LIN {X 0,Y 448.603,Z 481.559,A -85,B 0,C 180,E1 -8747.553,E2 -8747.553} C_VEL
LIN {X 0,Y 449.563,Z 469.193,A -85,B 0,C 180,E1 -8748.693,E2 -8748.693} C_VEL
LIN {X 0,Y 450.592,Z 455.729,A -85,B 0,C 180,E1 -8749.713,E2 -8749.713} C_VEL
LIN {X 0,Y 451.602,Z 440.797,A -85,B 0,C 180,E1 -8750.617,E2 -8750.617} C_VEL
LIN {X 0,Y 452.485,Z 425.824,A -85,B 0,C 180,E1 -8751.309,E2 -8751.309} C_VEL
LIN {X 0,Y 453.202,Z 410.38,A -85,B 0,C 180,E1 -8751.823,E2 -8751.823} C_VEL
LIN {X 0,Y 453.655,Z 394.686,A -85,B 0,C 180,E1 -8752.157,E2 -8752.157} C_VEL
LIN {X 0,Y 455.333,Z 264.862,A -85,B 0,C 180,E1 -8754.24,E2 -8754.24} C_VEL
LIN {X 0,Y 453.979,Z 251.014,A -85,B 0,C 180,E1 -8754.549,E2 -8754.549} C_VEL
LIN {X 0,Y 452.072,Z 236.66,A -85,B 0,C 180,E1 -8754.969,E2 -8754.969} C_VEL
LIN {X 0,Y 454.282,Z 211.093,A -85,B 0,C 180,E1 -8757.828,E2 -8757.828} C_VEL
LIN {X 0,Y 457.111,Z 186.417,A -85,B 0,C 180,E1 -8760.745,E2 -8760.745} C_VEL
LIN {X 0,Y 457.91,Z 180.659,A -85,B 0,C 180,E1 -8761.456,E2 -8761.456} C_VEL
LIN {X 0,Y 455.867,Z 172.549,A -85,B 0,C 180,E1 -8762.832,E2 -8762.832} C_VEL
LIN {X 0,Y 452.903,Z 163.172,A -85,B 0,C 180,E1 -8764.671,E2 -8764.671} C_VEL
LIN {X 0,Y 449.695,Z 154.889,A -85,B 0,C 180,E1 -8766.634,E2 -8766.634} C_VEL
LIN {X 0,Y 447.386,Z 149.256,A -85,B 0,C 180,E1 -8768.238,E2 -8768.238} C_VEL
LIN {X 0,Y 446.421,Z 146.504,A -85,B 0,C 180,E1 -8769.151,E2 -8769.151} C_VEL
LIN {X 0,Y 446.382,Z 146.509,A -85,B 0,C 180,E1 -8772.27,E2 -8772.27} C_VEL
LIN {X 0,Y 446.423,Z 146.505,A -85,B 0,C 180,E1 -8775.108,E2 -8775.108} C_VEL
LIN {X 0,Y 446.397,Z 146.505,A -85,B 0,C 180,E1 -8778.606,E2 -8778.606} C_VEL
LIN {X 0,Y 446.39,Z 146.508,A -85,B 0,C 180,E1 -8782.119,E2 -8782.119} C_VEL
LIN {X 0,Y 446.423,Z 146.505,A -85,B 0,C 180,E1 -8785.477,E2 -8785.477} C_VEL
LIN {X 0,Y 446.442,Z 146.59,A -85,B 0,C 180,E1 -8786.407,E2 -8786.407} C_VEL
LIN {X 0,Y 448.873,Z 153.492,A -85,B 0,C 180,E1 -8788.89,E2 -8788.89} C_VEL
LIN {X 0,Y 451.118,Z 160.8,A -85,B 0,C 180,E1 -8791.122,E2 -8791.122} C_VEL
LIN {X 0,Y 453.267,Z 168.747,A -85,B 0,C 180,E1 -8793.279,E2 -8793.279} C_VEL
LIN {X 0,Y 454.691,Z 176.225,A -85,B 0,C 180,E1 -8795.09,E2 -8795.09} C_VEL
LIN {X 0,Y 453.323,Z 189.363,A -85,B 0,C 180,E1 -8797.677,E2 -8797.677} C_VEL
LIN {X 0,Y 451.857,Z 205.223,A -85,B 0,C 180,E1 -8800.671,E2 -8800.671} C_VEL
LIN {X 0,Y 455.219,Z 218.827,A -85,B 0,C 180,E1 -8801.302,E2 -8801.302} C_VEL
LIN {X 0,Y 451.899,Z 307.293,A -85,B 0,C 180,E1 -8803.453,E2 -8803.453} C_VEL
LIN {X 0,Y 451.558,Z 325.184,A -85,B 0,C 180,E1 -8803.934,E2 -8803.934} C_VEL
LIN {X 0,Y 451.243,Z 338.258,A -85,B 0,C 180,E1 -8804.473,E2 -8804.473} C_VEL
LIN {X 0,Y 450.777,Z 351.293,A -85,B 0,C 180,E1 -8805.198,E2 -8805.198} C_VEL
LIN {X 0,Y 450.232,Z 362.94,A -85,B 0,C 180,E1 -8806.028,E2 -8806.028} C_VEL
LIN {X 0,Y 449.679,Z 373.95,A -85,B 0,C 180,E1 -8807.017,E2 -8807.017} C_VEL
LIN {X 0,Y 449.213,Z 383.222,A -85,B 0,C 180,E1 -8808.036,E2 -8808.036} C_VEL
LIN {X 0,Y 448.662,Z 391.778,A -85,B 0,C 180,E1 -8809.166,E2 -8809.166} C_VEL
LIN {X 0,Y 448.106,Z 400.134,A -85,B 0,C 180,E1 -8810.521,E2 -8810.521} C_VEL
LIN {X 0,Y 447.566,Z 406.817,A -85,B 0,C 180,E1 -8811.876,E2 -8811.876} C_VEL
LIN {X 0,Y 447.282,Z 412.123,A -85,B 0,C 180,E1 -8813.232,E2 -8813.232} C_VEL
LIN {X 0,Y 446.899,Z 416.261,A -85,B 0,C 180,E1 -8814.586,E2 -8814.586} C_VEL
LIN {X 0,Y 446.735,Z 418.408,A -85,B 0,C 180,E1 -8815.489,E2 -8815.489} C_VEL
LIN {X 0,Y 446.7,Z 420.094,A -85,B 0,C 180,E1 -8816.392,E2 -8816.392} C_VEL
LIN {X 0,Y 446.587,Z 421.324,A -85,B 0,C 180,E1 -8817.294,E2 -8817.294} C_VEL
LIN {X 0,Y 446.509,Z 422.142,A -85,B 0,C 180,E1 -8818.196,E2 -8818.196} C_VEL
LIN {X 0,Y 446.414,Z 422.565,A -85,B 0,C 180,E1 -8819.098,E2 -8819.098} C_VEL
LIN {X 0,Y 446.372,Z 422.567,A -85,B 0,C 180,E1 -8820,E2 -8820} C_VEL
LIN {X 0,Y 446.387,Z 422.116,A -85,B 0,C 180,E1 -8820.902,E2 -8820.902} C_VEL
LIN {X 0,Y 446.305,Z 421.284,A -85,B 0,C 180,E1 -8821.805,E2 -8821.805} C_VEL
LIN {X 0,Y 446.422,Z 420.025,A -85,B 0,C 180,E1 -8822.707,E2 -8822.707} C_VEL
LIN {X 0,Y 446.362,Z 417.34,A -85,B 0,C 180,E1 -8824.063,E2 -8824.063} C_VEL
LIN {X 0,Y 446.544,Z 413.61,A -85,B 0,C 180,E1 -8825.419,E2 -8825.419} C_VEL
LIN {X 0,Y 446.83,Z 408.619,A -85,B 0,C 180,E1 -8826.811,E2 -8826.811} C_VEL
LIN {X 0,Y 447.019,Z 402.697,A -85,B 0,C 180,E1 -8828.135,E2 -8828.135} C_VEL
LIN {X 0,Y 447.423,Z 395.107,A -85,B 0,C 180,E1 -8829.493,E2 -8829.493} C_VEL
LIN {X 0,Y 447.76,Z 385.722,A -85,B 0,C 180,E1 -8830.857,E2 -8830.857} C_VEL
LIN {X 0,Y 448.163,Z 376.127,A -85,B 0,C 180,E1 -8831.993,E2 -8831.993} C_VEL
LIN {X 0,Y 448.646,Z 365.513,A -85,B 0,C 180,E1 -8833.014,E2 -8833.014} C_VEL
LIN {X 0,Y 449.076,Z 352.8,A -85,B 0,C 180,E1 -8833.998,E2 -8833.998} C_VEL
LIN {X 0,Y 449.421,Z 340.82,A -85,B 0,C 180,E1 -8834.721,E2 -8834.721} C_VEL
LIN {X 0,Y 449.721,Z 326.89,A -85,B 0,C 180,E1 -8835.349,E2 -8835.349} C_VEL
LIN {X 0,Y 449.994,Z 313.038,A -85,B 0,C 180,E1 -8835.775,E2 -8835.775} C_VEL
LIN {X 0,Y 451.496,Z 214.96,A -85,B 0,C 180,E1 -8837.673,E2 -8837.673} C_VEL
LIN {X 0,Y 448.658,Z 199.549,A -85,B 0,C 180,E1 -8838.105,E2 -8838.105} C_VEL
LIN {X 0,Y 449.604,Z 180.934,A -85,B 0,C 180,E1 -8841.311,E2 -8841.311} C_VEL
LIN {X 0,Y 450.318,Z 165.889,A -85,B 0,C 180,E1 -8843.94,E2 -8843.94} C_VEL
LIN {X 0,Y 449.539,Z 160.406,A -85,B 0,C 180,E1 -8844.968,E2 -8844.968} C_VEL
LIN {X 0,Y 446.472,Z 146.498,A -85,B 0,C 180,E1 -8847.7,E2 -8847.7} C_VEL
LIN {X 0,Y 446.431,Z 146.5,A -85,B 0,C 180,E1 -8850.25,E2 -8850.25} C_VEL
LIN {X 0,Y 446.451,Z 146.501,A -85,B 0,C 180,E1 -8853.453,E2 -8853.453} C_VEL
LIN {X 0,Y 446.405,Z 146.503,A -85,B 0,C 180,E1 -8856.745,E2 -8856.745} C_VEL
LIN {X 0,Y 446.44,Z 146.491,A -85,B 0,C 180,E1 -8860.198,E2 -8860.198} C_VEL
LIN {X 0,Y 446.402,Z 146.498,A -85,B 0,C 180,E1 -8863.596,E2 -8863.596} C_VEL
LIN {X 0,Y 446.403,Z 146.503,A -85,B 0,C 180,E1 -8866.403,E2 -8866.403} C_VEL
LIN {X 0,Y 446.432,Z 146.501,A -85,B 0,C 180,E1 -8869.082,E2 -8869.082} C_VEL
LIN {X 0,Y 446.413,Z 146.503,A -85,B 0,C 180,E1 -8872.121,E2 -8872.121} C_VEL
LIN {X 0,Y 446.427,Z 146.503,A -85,B 0,C 180,E1 -8875.476,E2 -8875.476} C_VEL
LIN {X 0,Y 446.42,Z 146.503,A -85,B 0,C 180,E1 -8878.699,E2 -8878.699} C_VEL
LIN {X 0,Y 446.494,Z 146.615,A -85,B 0,C 180,E1 -8881.866,E2 -8881.866} C_VEL
LIN {X 0,Y 449.989,Z 159.891,A -85,B 0,C 180,E1 -8884.067,E2 -8884.067} C_VEL
LIN {X 0,Y 451.233,Z 164.799,A -85,B 0,C 180,E1 -8884.784,E2 -8884.784} C_VEL
LIN {X 0,Y 454.277,Z 173.036,A -85,B 0,C 180,E1 -8885.111,E2 -8885.111} C_VEL
LIN {X 0,Y 456.804,Z 184.373,A -85,B 0,C 180,E1 -8885.455,E2 -8885.455} C_VEL
LIN {X 0,Y 456.787,Z 190.412,A -85,B 0,C 180,E1 -8885.557,E2 -8885.557} C_VEL
LIN {X 0,Y 456.125,Z 196.262,A -85,B 0,C 180,E1 -8885.618,E2 -8885.618} C_VEL
LIN {X 0,Y 450.604,Z 215.327,A -85,B 0,C 180,E1 -8885.621,E2 -8885.621} C_VEL
LIN {X 0,Y 449.88,Z 221.18,A -85,B 0,C 180,E1 -8885.68,E2 -8885.68} C_VEL
LIN {X 0,Y 448.241,Z 331.634,A -85,B 0,C 180,E1 -8887.512,E2 -8887.512} C_VEL
LIN {X 0,Y 447.916,Z 346.746,A -85,B 0,C 180,E1 -8887.937,E2 -8887.937} C_VEL
LIN {X 0,Y 447.417,Z 359.567,A -85,B 0,C 180,E1 -8888.442,E2 -8888.442} C_VEL
LIN {X 0,Y 446.764,Z 373.298,A -85,B 0,C 180,E1 -8889.15,E2 -8889.15} C_VEL
LIN {X 0,Y 445.828,Z 387.352,A -85,B 0,C 180,E1 -8890.068,E2 -8890.068} C_VEL
LIN {X 0,Y 444.831,Z 400.144,A -85,B 0,C 180,E1 -8891.101,E2 -8891.101} C_VEL
LIN {X 0,Y 443.852,Z 412.557,A -85,B 0,C 180,E1 -8892.325,E2 -8892.325} C_VEL
LIN {X 0,Y 442.838,Z 423.693,A -85,B 0,C 180,E1 -8893.637,E2 -8893.637} C_VEL
LIN {X 0,Y 441.963,Z 433.554,A -85,B 0,C 180,E1 -8895.024,E2 -8895.024} C_VEL
LIN {X 0,Y 441.073,Z 442.905,A -85,B 0,C 180,E1 -8896.59,E2 -8896.59} C_VEL
LIN {X 0,Y 440.345,Z 451.156,A -85,B 0,C 180,E1 -8898.258,E2 -8898.258} C_VEL
LIN {X 0,Y 439.756,Z 457.752,A -85,B 0,C 180,E1 -8899.874,E2 -8899.874} C_VEL
LIN {X 0,Y 439.297,Z 463.848,A -85,B 0,C 180,E1 -8901.72,E2 -8901.72} C_VEL
LIN {X 0,Y 438.938,Z 468.563,A -85,B 0,C 180,E1 -8903.564,E2 -8903.564} C_VEL
LIN {X 0,Y 438.817,Z 472.01,A -85,B 0,C 180,E1 -8905.406,E2 -8905.406} C_VEL
LIN {X 0,Y 438.65,Z 474.293,A -85,B 0,C 180,E1 -8907.244,E2 -8907.244} C_VEL
LIN {X 0,Y 438.422,Z 475.467,A -85,B 0,C 180,E1 -8909.08,E2 -8909.08} C_VEL
LIN {X 0,Y 438.422,Z 475.482,A -85,B 0,C 180,E1 -8910.917,E2 -8910.917} C_VEL
LIN {X 0,Y 438.649,Z 474.369,A -85,B 0,C 180,E1 -8912.754,E2 -8912.754} C_VEL
LIN {X 0,Y 438.808,Z 472.151,A -85,B 0,C 180,E1 -8914.592,E2 -8914.592} C_VEL
LIN {X 0,Y 438.92,Z 468.778,A -85,B 0,C 180,E1 -8916.434,E2 -8916.434} C_VEL
LIN {X 0,Y 439.284,Z 464.136,A -85,B 0,C 180,E1 -8918.277,E2 -8918.277} C_VEL
LIN {X 0,Y 439.743,Z 458.109,A -85,B 0,C 180,E1 -8920.124,E2 -8920.124} C_VEL
LIN {X 0,Y 440.383,Z 450.519,A -85,B 0,C 180,E1 -8921.973,E2 -8921.973} C_VEL
LIN {X 0,Y 441.164,Z 442.089,A -85,B 0,C 180,E1 -8923.647,E2 -8923.647} C_VEL
LIN {X 0,Y 442.056,Z 432.628,A -85,B 0,C 180,E1 -8925.207,E2 -8925.207} C_VEL
LIN {X 0,Y 442.961,Z 422.624,A -85,B 0,C 180,E1 -8926.593,E2 -8926.593} C_VEL
LIN {X 0,Y 443.984,Z 410.668,A -85,B 0,C 180,E1 -8927.973,E2 -8927.973} C_VEL
LIN {X 0,Y 444.997,Z 398.609,A -85,B 0,C 180,E1 -8929.129,E2 -8929.129} C_VEL
LIN {X 0,Y 446.011,Z 385.476,A -85,B 0,C 180,E1 -8930.162,E2 -8930.162} C_VEL
LIN {X 0,Y 446.863,Z 370.893,A -85,B 0,C 180,E1 -8931.084,E2 -8931.084} C_VEL
LIN {X 0,Y 447.531,Z 356.049,A -85,B 0,C 180,E1 -8931.81,E2 -8931.81} C_VEL
LIN {X 0,Y 448.081,Z 341.166,A -85,B 0,C 180,E1 -8932.338,E2 -8932.338} C_VEL
LIN {X 0,Y 448.349,Z 327.58,A -85,B 0,C 180,E1 -8932.668,E2 -8932.668} C_VEL
LIN {X 0,Y 450.438,Z 185.764,A -85,B 0,C 180,E1 -8934.996,E2 -8934.996} C_VEL
LIN {X 0,Y 447.373,Z 172.856,A -85,B 0,C 180,E1 -8935.409,E2 -8935.409} C_VEL
LIN {X 0,Y 444.02,Z 164.852,A -85,B 0,C 180,E1 -8935.791,E2 -8935.791} C_VEL
LIN {X 0,Y 440.796,Z 152.391,A -85,B 0,C 180,E1 -8937.774,E2 -8937.774} C_VEL
LIN {X 0,Y 439.435,Z 147.373,A -85,B 0,C 180,E1 -8938.671,E2 -8938.671} C_VEL
LIN {X 0,Y 439.366,Z 147.373,A -85,B 0,C 180,E1 -8942.029,E2 -8942.029} C_VEL
LIN {X 0,Y 439.391,Z 147.38,A -85,B 0,C 180,E1 -8945.339,E2 -8945.339} C_VEL
LIN {X 0,Y 439.377,Z 147.377,A -85,B 0,C 180,E1 -8948.594,E2 -8948.594} C_VEL
LIN {X 0,Y 439.383,Z 147.367,A -85,B 0,C 180,E1 -8951.256,E2 -8951.256} C_VEL
LIN {X 0,Y 439.398,Z 147.37,A -85,B 0,C 180,E1 -8954.727,E2 -8954.727} C_VEL
LIN {X 0,Y 439.39,Z 147.374,A -85,B 0,C 180,E1 -8957.795,E2 -8957.795} C_VEL
LIN {X 0,Y 439.444,Z 147.367,A -85,B 0,C 180,E1 -8960.229,E2 -8960.229} C_VEL
LIN {X 0,Y 439.369,Z 147.378,A -85,B 0,C 180,E1 -8963.712,E2 -8963.712} C_VEL
LIN {X 0,Y 439.367,Z 147.38,A -85,B 0,C 180,E1 -8967.053,E2 -8967.053} C_VEL
LIN {X 0,Y 439.388,Z 147.365,A -85,B 0,C 180,E1 -8970.274,E2 -8970.274} C_VEL
LIN {X 0,Y 439.423,Z 147.369,A -85,B 0,C 180,E1 -8973.588,E2 -8973.588} C_VEL
LIN {X 0,Y 439.376,Z 147.372,A -85,B 0,C 180,E1 -8976.429,E2 -8976.429} C_VEL
LIN {X 0,Y 439.378,Z 147.373,A -85,B 0,C 180,E1 -8979.396,E2 -8979.396} C_VEL
LIN {X 0,Y 439.421,Z 147.366,A -85,B 0,C 180,E1 -8982.309,E2 -8982.309} C_VEL
LIN {X 0,Y 439.438,Z 147.367,A -85,B 0,C 180,E1 -8985.174,E2 -8985.174} C_VEL
LIN {X 0,Y 439.474,Z 147.356,A -85,B 0,C 180,E1 -8988.001,E2 -8988.001} C_VEL
LIN {X 0,Y 439.537,Z 147.353,A -85,B 0,C 180,E1 -8991.726,E2 -8991.726} C_VEL
LIN {X 0,Y 439.61,Z 147.338,A -85,B 0,C 180,E1 -8994.496,E2 -8994.496} C_VEL
LIN {X 0,Y 439.625,Z 147.346,A -85,B 0,C 180,E1 -8998.168,E2 -8998.168} C_VEL
LIN {X 0,Y 439.753,Z 147.319,A -85,B 0,C 180,E1 -9000,E2 -9000} C_VEL
LIN {X 0,Y 439.646,Z 147.347,A -85,B 0,C 180,E1 -9002.749,E2 -9002.749} C_VEL
LIN {X 0,Y 439.607,Z 147.338,A -85,B 0,C 180,E1 -9006.425,E2 -9006.425} C_VEL
LIN {X 0,Y 439.49,Z 147.36,A -85,B 0,C 180,E1 -9009.202,E2 -9009.202} C_VEL
LIN {X 0,Y 439.455,Z 147.355,A -85,B 0,C 180,E1 -9012.938,E2 -9012.938} C_VEL
LIN {X 0,Y 439.449,Z 147.37,A -85,B 0,C 180,E1 -9016.355,E2 -9016.355} C_VEL
LIN {X 0,Y 439.393,Z 147.364,A -85,B 0,C 180,E1 -9019.627,E2 -9019.627} C_VEL
LIN {X 0,Y 439.357,Z 147.379,A -85,B 0,C 180,E1 -9022.576,E2 -9022.576} C_VEL
LIN {X 0,Y 439.395,Z 147.369,A -85,B 0,C 180,E1 -9025.585,E2 -9025.585} C_VEL
LIN {X 0,Y 439.407,Z 147.368,A -85,B 0,C 180,E1 -9028.674,E2 -9028.674} C_VEL
LIN {X 0,Y 439.361,Z 147.382,A -85,B 0,C 180,E1 -9032.031,E2 -9032.031} C_VEL
LIN {X 0,Y 439.387,Z 147.373,A -85,B 0,C 180,E1 -9035.342,E2 -9035.342} C_VEL
LIN {X 0,Y 439.379,Z 147.364,A -85,B 0,C 180,E1 -9038.595,E2 -9038.595} C_VEL
LIN {X 0,Y 439.379,Z 147.359,A -85,B 0,C 180,E1 -9041.258,E2 -9041.258} C_VEL
LIN {X 0,Y 439.394,Z 147.376,A -85,B 0,C 180,E1 -9044.73,E2 -9044.73} C_VEL
LIN {X 0,Y 439.405,Z 147.377,A -85,B 0,C 180,E1 -9047.799,E2 -9047.799} C_VEL
LIN {X 0,Y 439.442,Z 147.372,A -85,B 0,C 180,E1 -9050.231,E2 -9050.231} C_VEL
LIN {X 0,Y 439.37,Z 147.376,A -85,B 0,C 180,E1 -9053.714,E2 -9053.714} C_VEL
LIN {X 0,Y 439.393,Z 147.429,A -85,B 0,C 180,E1 -9054.55,E2 -9054.55} C_VEL
LIN {X 0,Y 445.757,Z 168.464,A -85,B 0,C 180,E1 -9057.489,E2 -9057.489} C_VEL
LIN {X 0,Y 448.797,Z 178.964,A -85,B 0,C 180,E1 -9058.886,E2 -9058.886} C_VEL
LIN {X 0,Y 446.1,Z 212.955,A -85,B 0,C 180,E1 -9062.562,E2 -9062.562} C_VEL
LIN {X 0,Y 444.881,Z 231.94,A -85,B 0,C 180,E1 -9064.588,E2 -9064.588} C_VEL
LIN {X 0,Y 448.797,Z 263.831,A -85,B 0,C 180,E1 -9065.369,E2 -9065.369} C_VEL
LIN {X 0,Y 447.227,Z 382.055,A -85,B 0,C 180,E1 -9067.296,E2 -9067.296} C_VEL
LIN {X 0,Y 446.797,Z 404.556,A -85,B 0,C 180,E1 -9067.7,E2 -9067.7} C_VEL
LIN {X 0,Y 446.125,Z 419.902,A -85,B 0,C 180,E1 -9068.152,E2 -9068.152} C_VEL
LIN {X 0,Y 445.255,Z 434.727,A -85,B 0,C 180,E1 -9068.775,E2 -9068.775} C_VEL
LIN {X 0,Y 444.41,Z 448.229,A -85,B 0,C 180,E1 -9069.521,E2 -9069.521} C_VEL
LIN {X 0,Y 443.348,Z 461.563,A -85,B 0,C 180,E1 -9070.436,E2 -9070.436} C_VEL
LIN {X 0,Y 442.298,Z 475.142,A -85,B 0,C 180,E1 -9071.592,E2 -9071.592} C_VEL
LIN {X 0,Y 441.431,Z 486.843,A -85,B 0,C 180,E1 -9072.796,E2 -9072.796} C_VEL
LIN {X 0,Y 440.489,Z 498.759,A -85,B 0,C 180,E1 -9074.264,E2 -9074.264} C_VEL
LIN {X 0,Y 439.65,Z 509.698,A -85,B 0,C 180,E1 -9075.892,E2 -9075.892} C_VEL
LIN {X 0,Y 439.142,Z 518.621,A -85,B 0,C 180,E1 -9077.485,E2 -9077.485} C_VEL
LIN {X 0,Y 438.821,Z 527.349,A -85,B 0,C 180,E1 -9079.388,E2 -9079.388} C_VEL
LIN {X 0,Y 438.548,Z 534.198,A -85,B 0,C 180,E1 -9081.244,E2 -9081.244} C_VEL
LIN {X 0,Y 438.584,Z 539.573,A -85,B 0,C 180,E1 -9083.099,E2 -9083.099} C_VEL
LIN {X 0,Y 438.605,Z 542.66,A -85,B 0,C 180,E1 -9084.484,E2 -9084.484} C_VEL
LIN {X 0,Y 438.639,Z 545.687,A -85,B 0,C 180,E1 -9086.327,E2 -9086.327} C_VEL
LIN {X 0,Y 438.591,Z 547.489,A -85,B 0,C 180,E1 -9088.165,E2 -9088.165} C_VEL
LIN {X 0,Y 438.645,Z 548.109,A -85,B 0,C 180,E1 -9090.001,E2 -9090.001} C_VEL
LIN {X 0,Y 438.591,Z 547.489,A -85,B 0,C 180,E1 -9091.838,E2 -9091.838} C_VEL
LIN {X 0,Y 438.64,Z 545.687,A -85,B 0,C 180,E1 -9093.676,E2 -9093.676} C_VEL
LIN {X 0,Y 438.604,Z 542.653,A -85,B 0,C 180,E1 -9095.518,E2 -9095.518} C_VEL
LIN {X 0,Y 438.596,Z 538.327,A -85,B 0,C 180,E1 -9097.366,E2 -9097.366} C_VEL
LIN {X 0,Y 438.637,Z 532.608,A -85,B 0,C 180,E1 -9099.221,E2 -9099.221} C_VEL
LIN {X 0,Y 438.899,Z 525.353,A -85,B 0,C 180,E1 -9101.08,E2 -9101.08} C_VEL
LIN {X 0,Y 439.272,Z 517.378,A -85,B 0,C 180,E1 -9102.747,E2 -9102.747} C_VEL
LIN {X 0,Y 439.78,Z 508.222,A -85,B 0,C 180,E1 -9104.343,E2 -9104.343} C_VEL
LIN {X 0,Y 440.514,Z 498.723,A -85,B 0,C 180,E1 -9105.738,E2 -9105.738} C_VEL
LIN {X 0,Y 441.425,Z 486.832,A -85,B 0,C 180,E1 -9107.202,E2 -9107.202} C_VEL
LIN {X 0,Y 442.215,Z 476.257,A -85,B 0,C 180,E1 -9108.294,E2 -9108.294} C_VEL
LIN {X 0,Y 443.145,Z 464.364,A -85,B 0,C 180,E1 -9109.334,E2 -9109.334} C_VEL
LIN {X 0,Y 444.1,Z 451.678,A -85,B 0,C 180,E1 -9110.255,E2 -9110.255} C_VEL
LIN {X 0,Y 445.038,Z 437.98,A -85,B 0,C 180,E1 -9111.056,E2 -9111.056} C_VEL
LIN {X 0,Y 445.951,Z 423.205,A -85,B 0,C 180,E1 -9111.719,E2 -9111.719} C_VEL
LIN {X 0,Y 446.681,Z 408.798,A -85,B 0,C 180,E1 -9112.187,E2 -9112.187} C_VEL
LIN {X 0,Y 447.104,Z 392.425,A -85,B 0,C 180,E1 -9112.53,E2 -9112.53} C_VEL
LIN {X 0,Y 448.81,Z 263.796,A -85,B 0,C 180,E1 -9114.625,E2 -9114.625} C_VEL
LIN {X 0,Y 447.301,Z 249.61,A -85,B 0,C 180,E1 -9114.995,E2 -9114.995} C_VEL
LIN {X 0,Y 445.597,Z 236.028,A -85,B 0,C 180,E1 -9115.456,E2 -9115.456} C_VEL
LIN {X 0,Y 448.261,Z 208.763,A -85,B 0,C 180,E1 -9118.599,E2 -9118.599} C_VEL
LIN {X 0,Y 451.564,Z 183.576,A -85,B 0,C 180,E1 -9121.688,E2 -9121.688} C_VEL
LIN {X 0,Y 450.44,Z 178.248,A -85,B 0,C 180,E1 -9122.591,E2 -9122.591} C_VEL
LIN {X 0,Y 447.693,Z 168.89,A -85,B 0,C 180,E1 -9124.413,E2 -9124.413} C_VEL
LIN {X 0,Y 444.742,Z 160.784,A -85,B 0,C 180,E1 -9126.301,E2 -9126.301} C_VEL
LIN {X 0,Y 441.878,Z 153.645,A -85,B 0,C 180,E1 -9128.338,E2 -9128.338} C_VEL
LIN {X 0,Y 440.702,Z 150.674,A -85,B 0,C 180,E1 -9129.337,E2 -9129.337} C_VEL
LIN {X 0,Y 439.502,Z 148.11,A -85,B 0,C 180,E1 -9130.364,E2 -9130.364} C_VEL
LIN {X 0,Y 439.355,Z 147.384,A -85,B 0,C 180,E1 -9130.682,E2 -9130.682} C_VEL
LIN {X 0,Y 439.355,Z 147.385,A -85,B 0,C 180,E1 -9133.96,E2 -9133.96} C_VEL
LIN {X 0,Y 439.333,Z 147.385,A -85,B 0,C 180,E1 -9136.538,E2 -9136.538} C_VEL
LIN {X 0,Y 439.35,Z 147.385,A -85,B 0,C 180,E1 -9139.016,E2 -9139.016} C_VEL
LIN {X 0,Y 439.336,Z 147.386,A -85,B 0,C 180,E1 -9142.564,E2 -9142.564} C_VEL
LIN {X 0,Y 439.394,Z 147.383,A -85,B 0,C 180,E1 -9144.844,E2 -9144.844} C_VEL
LIN {X 0,Y 441.661,Z 153.659,A -85,B 0,C 180,E1 -9147.499,E2 -9147.499} C_VEL
LIN {X 0,Y 444.176,Z 161.248,A -85,B 0,C 180,E1 -9150.106,E2 -9150.106} C_VEL
LIN {X 0,Y 446.765,Z 170.807,A -85,B 0,C 180,E1 -9152.858,E2 -9152.858} C_VEL
LIN {X 0,Y 448.19,Z 178.084,A -85,B 0,C 180,E1 -9154.704,E2 -9154.704} C_VEL
LIN {X 0,Y 447.874,Z 182.864,A -85,B 0,C 180,E1 -9155.705,E2 -9155.705} C_VEL
LIN {X 0,Y 445.995,Z 199.55,A -85,B 0,C 180,E1 -9158.992,E2 -9158.992} C_VEL
LIN {X 0,Y 445.362,Z 205.7,A -85,B 0,C 180,E1 -9160.175,E2 -9160.175} C_VEL
LIN {X 0,Y 448.994,Z 220.092,A -85,B 0,C 180,E1 -9160.887,E2 -9160.887} C_VEL
LIN {X 0,Y 445.408,Z 307.337,A -85,B 0,C 180,E1 -9163.087,E2 -9163.087} C_VEL
LIN {X 0,Y 445.017,Z 325.15,A -85,B 0,C 180,E1 -9163.573,E2 -9163.573} C_VEL
LIN {X 0,Y 444.683,Z 338.473,A -85,B 0,C 180,E1 -9164.121,E2 -9164.121} C_VEL
LIN {X 0,Y 444.179,Z 352.044,A -85,B 0,C 180,E1 -9164.884,E2 -9164.884} C_VEL
LIN {X 0,Y 443.63,Z 362.994,A -85,B 0,C 180,E1 -9165.669,E2 -9165.669} C_VEL
LIN {X 0,Y 442.996,Z 374.478,A -85,B 0,C 180,E1 -9166.701,E2 -9166.701} C_VEL
LIN {X 0,Y 442.477,Z 382.9,A -85,B 0,C 180,E1 -9167.618,E2 -9167.618} C_VEL
LIN {X 0,Y 441.956,Z 391.655,A -85,B 0,C 180,E1 -9168.767,E2 -9168.767} C_VEL
LIN {X 0,Y 441.342,Z 400.238,A -85,B 0,C 180,E1 -9170.143,E2 -9170.143} C_VEL
LIN {X 0,Y 440.816,Z 406.936,A -85,B 0,C 180,E1 -9171.473,E2 -9171.473} C_VEL
LIN {X 0,Y 440.466,Z 411.781,A -85,B 0,C 180,E1 -9172.666,E2 -9172.666} C_VEL
LIN {X 0,Y 440.153,Z 416.234,A -85,B 0,C 180,E1 -9174.043,E2 -9174.043} C_VEL
LIN {X 0,Y 439.78,Z 419.59,A -85,B 0,C 180,E1 -9175.417,E2 -9175.417} C_VEL
LIN {X 0,Y 439.721,Z 421.247,A -85,B 0,C 180,E1 -9176.335,E2 -9176.335} C_VEL
LIN {X 0,Y 439.59,Z 422.448,A -85,B 0,C 180,E1 -9177.251,E2 -9177.251} C_VEL
LIN {X 0,Y 439.498,Z 423.24,A -85,B 0,C 180,E1 -9178.167,E2 -9178.167} C_VEL
LIN {X 0,Y 439.396,Z 423.633,A -85,B 0,C 180,E1 -9179.084,E2 -9179.084} C_VEL
LIN {X 0,Y 439.349,Z 423.593,A -85,B 0,C 180,E1 -9180,E2 -9180} C_VEL
LIN {X 0,Y 439.364,Z 423.107,A -85,B 0,C 180,E1 -9180.917,E2 -9180.917} C_VEL
LIN {X 0,Y 439.281,Z 422.241,A -85,B 0,C 180,E1 -9181.834,E2 -9181.834} C_VEL
LIN {X 0,Y 439.399,Z 420.951,A -85,B 0,C 180,E1 -9182.75,E2 -9182.75} C_VEL
LIN {X 0,Y 439.342,Z 418.203,A -85,B 0,C 180,E1 -9184.128,E2 -9184.128} C_VEL
LIN {X 0,Y 439.541,Z 414.405,A -85,B 0,C 180,E1 -9185.505,E2 -9185.505} C_VEL
LIN {X 0,Y 439.825,Z 409.491,A -85,B 0,C 180,E1 -9186.883,E2 -9186.883} C_VEL
LIN {X 0,Y 440.015,Z 403.33,A -85,B 0,C 180,E1 -9188.265,E2 -9188.265} C_VEL
LIN {X 0,Y 440.433,Z 395.636,A -85,B 0,C 180,E1 -9189.645,E2 -9189.645} C_VEL
LIN {X 0,Y 440.812,Z 386.148,A -85,B 0,C 180,E1 -9191.03,E2 -9191.03} C_VEL
LIN {X 0,Y 441.243,Z 376.418,A -85,B 0,C 180,E1 -9192.184,E2 -9192.184} C_VEL
LIN {X 0,Y 441.738,Z 365.657,A -85,B 0,C 180,E1 -9193.221,E2 -9193.221} C_VEL
LIN {X 0,Y 442.163,Z 352.949,A -85,B 0,C 180,E1 -9194.209,E2 -9194.209} C_VEL
LIN {X 0,Y 442.535,Z 340.518,A -85,B 0,C 180,E1 -9194.956,E2 -9194.956} C_VEL
LIN {X 0,Y 442.84,Z 327.041,A -85,B 0,C 180,E1 -9195.564,E2 -9195.564} C_VEL
LIN {X 0,Y 443.102,Z 314.172,A -85,B 0,C 180,E1 -9195.967,E2 -9195.967} C_VEL
LIN {X 0,Y 444.701,Z 216.012,A -85,B 0,C 180,E1 -9197.919,E2 -9197.919} C_VEL
LIN {X 0,Y 441.787,Z 199.752,A -85,B 0,C 180,E1 -9198.389,E2 -9198.389} C_VEL
LIN {X 0,Y 442.728,Z 180.989,A -85,B 0,C 180,E1 -9201.659,E2 -9201.659} C_VEL
LIN {X 0,Y 443.445,Z 167.249,A -85,B 0,C 180,E1 -9204.086,E2 -9204.086} C_VEL
LIN {X 0,Y 442.575,Z 161.607,A -85,B 0,C 180,E1 -9205.155,E2 -9205.155} C_VEL
LIN {X 0,Y 439.425,Z 147.375,A -85,B 0,C 180,E1 -9207.985,E2 -9207.985} C_VEL
LIN {X 0,Y 439.365,Z 147.381,A -85,B 0,C 180,E1 -9210.788,E2 -9210.788} C_VEL
LIN {X 0,Y 439.392,Z 147.376,A -85,B 0,C 180,E1 -9214.043,E2 -9214.043} C_VEL
LIN {X 0,Y 439.351,Z 147.383,A -85,B 0,C 180,E1 -9216.886,E2 -9216.886} C_VEL
LIN {X 0,Y 439.381,Z 147.37,A -85,B 0,C 180,E1 -9219.845,E2 -9219.845} C_VEL
LIN {X 0,Y 439.375,Z 147.379,A -85,B 0,C 180,E1 -9222.625,E2 -9222.625} C_VEL
LIN {X 0,Y 439.404,Z 147.378,A -85,B 0,C 180,E1 -9225.27,E2 -9225.27} C_VEL
LIN {X 0,Y 439.393,Z 147.38,A -85,B 0,C 180,E1 -9228.743,E2 -9228.743} C_VEL
LIN {X 0,Y 439.378,Z 147.38,A -85,B 0,C 180,E1 -9231.607,E2 -9231.607} C_VEL
LIN {X 0,Y 439.401,Z 147.378,A -85,B 0,C 180,E1 -9234.843,E2 -9234.843} C_VEL
LIN {X 0,Y 439.376,Z 147.382,A -85,B 0,C 180,E1 -9238.139,E2 -9238.139} C_VEL
LIN {X 0,Y 439.456,Z 147.569,A -85,B 0,C 180,E1 -9241.464,E2 -9241.464} C_VEL
LIN {X 0,Y 442.925,Z 160.318,A -85,B 0,C 180,E1 -9243.622,E2 -9243.622} C_VEL
LIN {X 0,Y 444.204,Z 165.287,A -85,B 0,C 180,E1 -9244.356,E2 -9244.356} C_VEL
LIN {X 0,Y 447.929,Z 174.682,A -85,B 0,C 180,E1 -9244.754,E2 -9244.754} C_VEL
LIN {X 0,Y 450.346,Z 184.868,A -85,B 0,C 180,E1 -9245.079,E2 -9245.079} C_VEL
LIN {X 0,Y 449.88,Z 221.18,A -85,B 0,C 180,E1 -9245.68,E2 -9245.68} C_VEL
LIN {X 0,Y 449.137,Z 227.036,A -85,B 0,C 180,E1 -9245.737,E2 -9245.737} C_VEL
LIN {X 0,Y 443.587,Z 246.092,A -85,B 0,C 180,E1 -9245.741,E2 -9245.741} C_VEL
LIN {X 0,Y 443.038,Z 251.933,A -85,B 0,C 180,E1 -9245.811,E2 -9245.811} C_VEL
LIN {X 0,Y 441.718,Z 332.149,A -85,B 0,C 180,E1 -9247.161,E2 -9247.161} C_VEL
LIN {X 0,Y 441.38,Z 347.128,A -85,B 0,C 180,E1 -9247.587,E2 -9247.587} C_VEL
LIN {X 0,Y 440.844,Z 360.271,A -85,B 0,C 180,E1 -9248.111,E2 -9248.111} C_VEL
LIN {X 0,Y 440.164,Z 373.865,A -85,B 0,C 180,E1 -9248.822,E2 -9248.822} C_VEL
LIN {X 0,Y 439.193,Z 387.924,A -85,B 0,C 180,E1 -9249.753,E2 -9249.753} C_VEL
LIN {X 0,Y 438.152,Z 400.72,A -85,B 0,C 180,E1 -9250.802,E2 -9250.802} C_VEL
LIN {X 0,Y 437.098,Z 413.215,A -85,B 0,C 180,E1 -9252.052,E2 -9252.052} C_VEL
LIN {X 0,Y 436.058,Z 424.273,A -85,B 0,C 180,E1 -9253.376,E2 -9253.376} C_VEL
LIN {X 0,Y 435.11,Z 434.138,A -85,B 0,C 180,E1 -9254.782,E2 -9254.782} C_VEL
LIN {X 0,Y 434.145,Z 443.786,A -85,B 0,C 180,E1 -9256.427,E2 -9256.427} C_VEL
LIN {X 0,Y 433.41,Z 451.741,A -85,B 0,C 180,E1 -9258.067,E2 -9258.067} C_VEL
LIN {X 0,Y 432.782,Z 458.337,A -85,B 0,C 180,E1 -9259.709,E2 -9259.709} C_VEL
LIN {X 0,Y 432.299,Z 464.432,A -85,B 0,C 180,E1 -9261.585,E2 -9261.585} C_VEL
LIN {X 0,Y 431.912,Z 469.148,A -85,B 0,C 180,E1 -9263.459,E2 -9263.459} C_VEL
LIN {X 0,Y 431.772,Z 472.595,A -85,B 0,C 180,E1 -9265.331,E2 -9265.331} C_VEL
LIN {X 0,Y 431.604,Z 474.876,A -85,B 0,C 180,E1 -9267.199,E2 -9267.199} C_VEL
LIN {X 0,Y 431.361,Z 476.05,A -85,B 0,C 180,E1 -9269.065,E2 -9269.065} C_VEL
LIN {X 0,Y 431.36,Z 476.066,A -85,B 0,C 180,E1 -9270.932,E2 -9270.932} C_VEL
LIN {X 0,Y 431.603,Z 474.951,A -85,B 0,C 180,E1 -9272.799,E2 -9272.799} C_VEL
LIN {X 0,Y 431.762,Z 472.735,A -85,B 0,C 180,E1 -9274.667,E2 -9274.667} C_VEL
LIN {X 0,Y 431.893,Z 469.361,A -85,B 0,C 180,E1 -9276.539,E2 -9276.539} C_VEL
LIN {X 0,Y 432.29,Z 464.717,A -85,B 0,C 180,E1 -9278.412,E2 -9278.412} C_VEL
LIN {X 0,Y 432.769,Z 458.691,A -85,B 0,C 180,E1 -9280.289,E2 -9280.289} C_VEL
LIN {X 0,Y 433.447,Z 451.1,A -85,B 0,C 180,E1 -9282.167,E2 -9282.167} C_VEL
LIN {X 0,Y 434.252,Z 442.936,A -85,B 0,C 180,E1 -9283.82,E2 -9283.82} C_VEL
LIN {X 0,Y 435.21,Z 433.206,A -85,B 0,C 180,E1 -9285.452,E2 -9285.452} C_VEL
LIN {X 0,Y 436.187,Z 423.197,A -85,B 0,C 180,E1 -9286.858,E2 -9286.858} C_VEL
LIN {X 0,Y 437.227,Z 411.494,A -85,B 0,C 180,E1 -9288.234,E2 -9288.234} C_VEL
LIN {X 0,Y 438.31,Z 399.175,A -85,B 0,C 180,E1 -9289.432,E2 -9289.432} C_VEL
LIN {X 0,Y 439.389,Z 386.034,A -85,B 0,C 180,E1 -9290.479,E2 -9290.479} C_VEL
LIN {X 0,Y 440.287,Z 371.441,A -85,B 0,C 180,E1 -9291.415,E2 -9291.415} C_VEL
LIN {X 0,Y 440.975,Z 356.391,A -85,B 0,C 180,E1 -9292.159,E2 -9292.159} C_VEL
LIN {X 0,Y 441.562,Z 341.131,A -85,B 0,C 180,E1 -9292.702,E2 -9292.702} C_VEL
LIN {X 0,Y 441.874,Z 326.059,A -85,B 0,C 180,E1 -9293.056,E2 -9293.056} C_VEL
LIN {X 0,Y 444.016,Z 187.556,A -85,B 0,C 180,E1 -9295.359,E2 -9295.359} C_VEL
LIN {X 0,Y 443.442,Z 183.871,A -85,B 0,C 180,E1 -9295.46,E2 -9295.46} C_VEL
LIN {X 0,Y 441.142,Z 175.179,A -85,B 0,C 180,E1 -9295.76,E2 -9295.76} C_VEL
LIN {X 0,Y 437.026,Z 165.534,A -85,B 0,C 180,E1 -9296.213,E2 -9296.213} C_VEL
LIN {X 0,Y 434.056,Z 154.305,A -85,B 0,C 180,E1 -9298.004,E2 -9298.004} C_VEL
LIN {X 0,Y 432.376,Z 148.253,A -85,B 0,C 180,E1 -9299.066,E2 -9299.066} C_VEL
LIN {X 0,Y 432.319,Z 148.251,A -85,B 0,C 180,E1 -9302.442,E2 -9302.442} C_VEL
LIN {X 0,Y 432.341,Z 148.259,A -85,B 0,C 180,E1 -9305.631,E2 -9305.631} C_VEL
LIN {X 0,Y 432.339,Z 148.254,A -85,B 0,C 180,E1 -9308.714,E2 -9308.714} C_VEL
LIN {X 0,Y 432.357,Z 148.252,A -85,B 0,C 180,E1 -9311.792,E2 -9311.792} C_VEL
LIN {X 0,Y 432.333,Z 148.249,A -85,B 0,C 180,E1 -9314.345,E2 -9314.345} C_VEL
LIN {X 0,Y 432.313,Z 148.258,A -85,B 0,C 180,E1 -9317.014,E2 -9317.014} C_VEL
LIN {X 0,Y 432.349,Z 148.252,A -85,B 0,C 180,E1 -9319.816,E2 -9319.816} C_VEL
LIN {X 0,Y 432.309,Z 148.261,A -85,B 0,C 180,E1 -9323.022,E2 -9323.022} C_VEL
LIN {X 0,Y 432.351,Z 148.248,A -85,B 0,C 180,E1 -9325.995,E2 -9325.995} C_VEL
LIN {X 0,Y 432.387,Z 148.237,A -85,B 0,C 180,E1 -9329.743,E2 -9329.743} C_VEL
LIN {X 0,Y 432.39,Z 148.247,A -85,B 0,C 180,E1 -9333.372,E2 -9333.372} C_VEL
LIN {X 0,Y 432.361,Z 148.244,A -85,B 0,C 180,E1 -9336.023,E2 -9336.023} C_VEL
LIN {X 0,Y 432.34,Z 148.254,A -85,B 0,C 180,E1 -9339.045,E2 -9339.045} C_VEL
LIN {X 0,Y 432.367,Z 148.243,A -85,B 0,C 180,E1 -9342.011,E2 -9342.011} C_VEL
LIN {X 0,Y 432.386,Z 148.249,A -85,B 0,C 180,E1 -9344.926,E2 -9344.926} C_VEL
LIN {X 0,Y 432.449,Z 148.231,A -85,B 0,C 180,E1 -9347.803,E2 -9347.803} C_VEL
LIN {X 0,Y 432.481,Z 148.232,A -85,B 0,C 180,E1 -9351.59,E2 -9351.59} C_VEL
LIN {X 0,Y 432.587,Z 148.212,A -85,B 0,C 180,E1 -9354.406,E2 -9354.406} C_VEL
LIN {X 0,Y 432.595,Z 148.221,A -85,B 0,C 180,E1 -9358.138,E2 -9358.138} C_VEL
LIN {X 0,Y 432.723,Z 148.194,A -85,B 0,C 180,E1 -9360,E2 -9360} C_VEL
LIN {X 0,Y 432.595,Z 148.225,A -85,B 0,C 180,E1 -9362.794,E2 -9362.794} C_VEL
LIN {X 0,Y 432.561,Z 148.215,A -85,B 0,C 180,E1 -9366.53,E2 -9366.53} C_VEL
LIN {X 0,Y 432.433,Z 148.239,A -85,B 0,C 180,E1 -9369.353,E2 -9369.353} C_VEL
LIN {X 0,Y 432.419,Z 148.231,A -85,B 0,C 180,E1 -9372.804,E2 -9372.804} C_VEL
LIN {X 0,Y 432.412,Z 148.246,A -85,B 0,C 180,E1 -9376.484,E2 -9376.484} C_VEL
LIN {X 0,Y 432.33,Z 148.245,A -85,B 0,C 180,E1 -9379.961,E2 -9379.961} C_VEL
LIN {X 0,Y 432.31,Z 148.253,A -85,B 0,C 180,E1 -9382.965,E2 -9382.965} C_VEL
LIN {X 0,Y 432.354,Z 148.249,A -85,B 0,C 180,E1 -9386.033,E2 -9386.033} C_VEL
LIN {X 0,Y 432.332,Z 148.246,A -85,B 0,C 180,E1 -9389.188,E2 -9389.188} C_VEL
LIN {X 0,Y 432.313,Z 148.259,A -85,B 0,C 180,E1 -9392.444,E2 -9392.444} C_VEL
LIN {X 0,Y 432.336,Z 148.253,A -85,B 0,C 180,E1 -9395.633,E2 -9395.633} C_VEL
LIN {X 0,Y 432.341,Z 148.239,A -85,B 0,C 180,E1 -9398.717,E2 -9398.717} C_VEL
LIN {X 0,Y 432.324,Z 148.24,A -85,B 0,C 180,E1 -9401.798,E2 -9401.798} C_VEL
LIN {X 0,Y 432.37,Z 148.253,A -85,B 0,C 180,E1 -9405.66,E2 -9405.66} C_VEL
LIN {X 0,Y 432.366,Z 148.254,A -85,B 0,C 180,E1 -9408.393,E2 -9408.393} C_VEL
LIN {X 0,Y 432.344,Z 148.253,A -85,B 0,C 180,E1 -9411.853,E2 -9411.853} C_VEL
LIN {X 0,Y 432.337,Z 148.311,A -85,B 0,C 180,E1 -9414.148,E2 -9414.148} C_VEL
LIN {X 0,Y 438.892,Z 169.95,A -85,B 0,C 180,E1 -9417.227,E2 -9417.227} C_VEL
LIN {X 0,Y 441.899,Z 180.148,A -85,B 0,C 180,E1 -9418.612,E2 -9418.612} C_VEL
LIN {X 0,Y 441.61,Z 185.79,A -85,B 0,C 180,E1 -9419.247,E2 -9419.247} C_VEL
LIN {X 0,Y 439.179,Z 215.277,A -85,B 0,C 180,E1 -9422.481,E2 -9422.481} C_VEL
LIN {X 0,Y 438.125,Z 230.62,A -85,B 0,C 180,E1 -9424.147,E2 -9424.147} C_VEL
LIN {X 0,Y 442.316,Z 264.023,A -85,B 0,C 180,E1 -9424.995,E2 -9424.995} C_VEL
LIN {X 0,Y 440.877,Z 370.816,A -85,B 0,C 180,E1 -9426.764,E2 -9426.764} C_VEL
LIN {X 0,Y 440.283,Z 402.925,A -85,B 0,C 180,E1 -9427.321,E2 -9427.321} C_VEL
LIN {X 0,Y 439.607,Z 418.611,A -85,B 0,C 180,E1 -9427.78,E2 -9427.78} C_VEL
LIN {X 0,Y 438.694,Z 433.047,A -85,B 0,C 180,E1 -9428.38,E2 -9428.38} C_VEL
LIN {X 0,Y 437.699,Z 447.716,A -85,B 0,C 180,E1 -9429.196,E2 -9429.196} C_VEL
LIN {X 0,Y 436.582,Z 460.989,A -85,B 0,C 180,E1 -9430.121,E2 -9430.121} C_VEL
LIN {X 0,Y 435.506,Z 474.565,A -85,B 0,C 180,E1 -9431.294,E2 -9431.294} C_VEL
LIN {X 0,Y 434.564,Z 486.126,A -85,B 0,C 180,E1 -9432.5,E2 -9432.5} C_VEL
LIN {X 0,Y 433.643,Z 496.387,A -85,B 0,C 180,E1 -9433.767,E2 -9433.767} C_VEL
LIN {X 0,Y 432.867,Z 506.157,A -85,B 0,C 180,E1 -9435.185,E2 -9435.185} C_VEL
LIN {X 0,Y 432.26,Z 515.754,A -85,B 0,C 180,E1 -9436.844,E2 -9436.844} C_VEL
LIN {X 0,Y 431.815,Z 523.741,A -85,B 0,C 180,E1 -9438.501,E2 -9438.501} C_VEL
LIN {X 0,Y 431.546,Z 530.375,A -85,B 0,C 180,E1 -9440.155,E2 -9440.155} C_VEL
LIN {X 0,Y 431.474,Z 536.474,A -85,B 0,C 180,E1 -9442.043,E2 -9442.043} C_VEL
LIN {X 0,Y 431.52,Z 540.081,A -85,B 0,C 180,E1 -9443.455,E2 -9443.455} C_VEL
LIN {X 0,Y 431.501,Z 543.74,A -85,B 0,C 180,E1 -9445.33,E2 -9445.33} C_VEL
LIN {X 0,Y 431.607,Z 546.158,A -85,B 0,C 180,E1 -9447.201,E2 -9447.201} C_VEL
LIN {X 0,Y 431.552,Z 547.365,A -85,B 0,C 180,E1 -9449.068,E2 -9449.068} C_VEL
LIN {X 0,Y 431.532,Z 547.364,A -85,B 0,C 180,E1 -9450.934,E2 -9450.934} C_VEL
LIN {X 0,Y 431.61,Z 546.158,A -85,B 0,C 180,E1 -9452.801,E2 -9452.801} C_VEL
LIN {X 0,Y 431.489,Z 543.736,A -85,B 0,C 180,E1 -9454.672,E2 -9454.672} C_VEL
LIN {X 0,Y 431.522,Z 540.069,A -85,B 0,C 180,E1 -9456.547,E2 -9456.547} C_VEL
LIN {X 0,Y 431.516,Z 535.058,A -85,B 0,C 180,E1 -9458.43,E2 -9458.43} C_VEL
LIN {X 0,Y 431.67,Z 528.593,A -85,B 0,C 180,E1 -9460.318,E2 -9460.318} C_VEL
LIN {X 0,Y 431.973,Z 520.477,A -85,B 0,C 180,E1 -9462.212,E2 -9462.212} C_VEL
LIN {X 0,Y 432.502,Z 511.832,A -85,B 0,C 180,E1 -9463.869,E2 -9463.869} C_VEL
LIN {X 0,Y 433.291,Z 501.434,A -85,B 0,C 180,E1 -9465.524,E2 -9465.524} C_VEL
LIN {X 0,Y 434.222,Z 489.776,A -85,B 0,C 180,E1 -9467.064,E2 -9467.064} C_VEL
LIN {X 0,Y 435.184,Z 478.039,A -85,B 0,C 180,E1 -9468.357,E2 -9468.357} C_VEL
LIN {X 0,Y 436.256,Z 465.216,A -85,B 0,C 180,E1 -9469.53,E2 -9469.53} C_VEL
LIN {X 0,Y 437.406,Z 451.104,A -85,B 0,C 180,E1 -9470.579,E2 -9470.579} C_VEL
LIN {X 0,Y 438.392,Z 437.414,A -85,B 0,C 180,E1 -9471.391,E2 -9471.391} C_VEL
LIN {X 0,Y 439.348,Z 422.562,A -85,B 0,C 180,E1 -9472.067,E2 -9472.067} C_VEL
LIN {X 0,Y 440.099,Z 408.268,A -85,B 0,C 180,E1 -9472.537,E2 -9472.537} C_VEL
LIN {X 0,Y 440.539,Z 391.941,A -85,B 0,C 180,E1 -9472.885,E2 -9472.885} C_VEL
LIN {X 0,Y 442.385,Z 265.411,A -85,B 0,C 180,E1 -9474.971,E2 -9474.971} C_VEL
LIN {X 0,Y 440.716,Z 247.523,A -85,B 0,C 180,E1 -9475.514,E2 -9475.514} C_VEL
LIN {X 0,Y 439.18,Z 235.471,A -85,B 0,C 180,E1 -9475.962,E2 -9475.962} C_VEL
LIN {X 0,Y 442.243,Z 207.286,A -85,B 0,C 180,E1 -9479.313,E2 -9479.313} C_VEL
LIN {X 0,Y 445.232,Z 186.603,A -85,B 0,C 180,E1 -9481.925,E2 -9481.925} C_VEL
LIN {X 0,Y 445.184,Z 184.816,A -85,B 0,C 180,E1 -9482.196,E2 -9482.196} C_VEL
LIN {X 0,Y 442.48,Z 174.811,A -85,B 0,C 180,E1 -9484.116,E2 -9484.116} C_VEL
LIN {X 0,Y 439.811,Z 166.93,A -85,B 0,C 180,E1 -9485.912,E2 -9485.912} C_VEL
LIN {X 0,Y 436.972,Z 159.453,A -85,B 0,C 180,E1 -9487.993,E2 -9487.993} C_VEL
LIN {X 0,Y 435.461,Z 155.777,A -85,B 0,C 180,E1 -9489.224,E2 -9489.224} C_VEL
LIN {X 0,Y 433.502,Z 151.361,A -85,B 0,C 180,E1 -9491.074,E2 -9491.074} C_VEL
LIN {X 0,Y 432.302,Z 148.262,A -85,B 0,C 180,E1 -9492.779,E2 -9492.779} C_VEL
LIN {X 0,Y 432.334,Z 148.258,A -85,B 0,C 180,E1 -9495.666,E2 -9495.666} C_VEL
LIN {X 0,Y 432.306,Z 148.261,A -85,B 0,C 180,E1 -9498.403,E2 -9498.403} C_VEL
LIN {X 0,Y 432.321,Z 148.261,A -85,B 0,C 180,E1 -9501.848,E2 -9501.848} C_VEL
LIN {X 0,Y 432.313,Z 148.397,A -85,B 0,C 180,E1 -9502.806,E2 -9502.806} C_VEL
LIN {X 0,Y 433.786,Z 151.892,A -85,B 0,C 180,E1 -9504.89,E2 -9504.89} C_VEL
LIN {X 0,Y 435.871,Z 157.792,A -85,B 0,C 180,E1 -9507.487,E2 -9507.487} C_VEL
LIN {X 0,Y 438.152,Z 164.949,A -85,B 0,C 180,E1 -9510.017,E2 -9510.017} C_VEL
LIN {X 0,Y 440.292,Z 172.967,A -85,B 0,C 180,E1 -9512.426,E2 -9512.426} C_VEL
LIN {X 0,Y 441.872,Z 181.138,A -85,B 0,C 180,E1 -9514.568,E2 -9514.568} C_VEL
LIN {X 0,Y 440.983,Z 189.261,A -85,B 0,C 180,E1 -9516.271,E2 -9516.271} C_VEL
LIN {X 0,Y 438.988,Z 206.31,A -85,B 0,C 180,E1 -9519.653,E2 -9519.653} C_VEL
LIN {X 0,Y 442.679,Z 220.856,A -85,B 0,C 180,E1 -9520.423,E2 -9520.423} C_VEL
LIN {X 0,Y 442.458,Z 229.975,A -85,B 0,C 180,E1 -9520.685,E2 -9520.685} C_VEL
LIN {X 0,Y 438.828,Z 312.307,A -85,B 0,C 180,E1 -9522.826,E2 -9522.826} C_VEL
LIN {X 0,Y 438.504,Z 327.121,A -85,B 0,C 180,E1 -9523.262,E2 -9523.262} C_VEL
LIN {X 0,Y 438.115,Z 340.014,A -85,B 0,C 180,E1 -9523.816,E2 -9523.816} C_VEL
LIN {X 0,Y 437.512,Z 354.169,A -85,B 0,C 180,E1 -9524.639,E2 -9524.639} C_VEL
LIN {X 0,Y 436.857,Z 366.316,A -85,B 0,C 180,E1 -9525.561,E2 -9525.561} C_VEL
LIN {X 0,Y 436.202,Z 377.343,A -85,B 0,C 180,E1 -9526.608,E2 -9526.608} C_VEL
LIN {X 0,Y 435.691,Z 386.385,A -85,B 0,C 180,E1 -9527.659,E2 -9527.659} C_VEL
LIN {X 0,Y 435.039,Z 394.753,A -85,B 0,C 180,E1 -9528.822,E2 -9528.822} C_VEL
LIN {X 0,Y 434.396,Z 402.906,A -85,B 0,C 180,E1 -9530.219,E2 -9530.219} C_VEL
LIN {X 0,Y 433.793,Z 409.477,A -85,B 0,C 180,E1 -9531.616,E2 -9531.616} C_VEL
LIN {X 0,Y 433.43,Z 414.669,A -85,B 0,C 180,E1 -9533.015,E2 -9533.015} C_VEL
LIN {X 0,Y 432.978,Z 418.711,A -85,B 0,C 180,E1 -9534.411,E2 -9534.411} C_VEL
LIN {X 0,Y 432.82,Z 420.801,A -85,B 0,C 180,E1 -9535.343,E2 -9535.343} C_VEL
LIN {X 0,Y 432.742,Z 422.411,A -85,B 0,C 180,E1 -9536.275,E2 -9536.275} C_VEL
LIN {X 0,Y 432.592,Z 423.583,A -85,B 0,C 180,E1 -9537.206,E2 -9537.206} C_VEL
LIN {X 0,Y 432.489,Z 424.344,A -85,B 0,C 180,E1 -9538.138,E2 -9538.138} C_VEL
LIN {X 0,Y 432.38,Z 424.706,A -85,B 0,C 180,E1 -9539.069,E2 -9539.069} C_VEL
LIN {X 0,Y 432.325,Z 424.62,A -85,B 0,C 180,E1 -9540,E2 -9540} C_VEL
LIN {X 0,Y 432.341,Z 424.101,A -85,B 0,C 180,E1 -9540.932,E2 -9540.932} C_VEL
LIN {X 0,Y 432.258,Z 423.2,A -85,B 0,C 180,E1 -9541.864,E2 -9541.864} C_VEL
LIN {X 0,Y 432.376,Z 421.869,A -85,B 0,C 180,E1 -9542.795,E2 -9542.795} C_VEL
LIN {X 0,Y 432.322,Z 419.057,A -85,B 0,C 180,E1 -9544.195,E2 -9544.195} C_VEL
LIN {X 0,Y 432.54,Z 415.187,A -85,B 0,C 180,E1 -9545.595,E2 -9545.595} C_VEL
LIN {X 0,Y 432.827,Z 410.197,A -85,B 0,C 180,E1 -9546.995,E2 -9546.995} C_VEL
LIN {X 0,Y 433.019,Z 403.935,A -85,B 0,C 180,E1 -9548.399,E2 -9548.399} C_VEL
LIN {X 0,Y 433.461,Z 396.139,A -85,B 0,C 180,E1 -9549.802,E2 -9549.802} C_VEL
LIN {X 0,Y 433.859,Z 386.546,A -85,B 0,C 180,E1 -9551.209,E2 -9551.209} C_VEL
LIN {X 0,Y 434.361,Z 375.54,A -85,B 0,C 180,E1 -9552.498,E2 -9552.498} C_VEL
LIN {X 0,Y 434.884,Z 364.417,A -85,B 0,C 180,E1 -9553.552,E2 -9553.552} C_VEL
LIN {X 0,Y 435.241,Z 353.471,A -85,B 0,C 180,E1 -9554.397,E2 -9554.397} C_VEL
LIN {X 0,Y 435.662,Z 340.14,A -85,B 0,C 180,E1 -9555.197,E2 -9555.197} C_VEL
LIN {X 0,Y 435.962,Z 327.085,A -85,B 0,C 180,E1 -9555.786,E2 -9555.786} C_VEL
LIN {X 0,Y 436.237,Z 313.827,A -85,B 0,C 180,E1 -9556.195,E2 -9556.195} C_VEL
LIN {X 0,Y 437.83,Z 216.462,A -85,B 0,C 180,E1 -9558.181,E2 -9558.181} C_VEL
LIN {X 0,Y 434.891,Z 200.033,A -85,B 0,C 180,E1 -9558.665,E2 -9558.665} C_VEL
LIN {X 0,Y 435.837,Z 182.383,A -85,B 0,C 180,E1 -9561.77,E2 -9561.77} C_VEL
LIN {X 0,Y 436.572,Z 168.595,A -85,B 0,C 180,E1 -9564.237,E2 -9564.237} C_VEL
LIN {X 0,Y 435.457,Z 161.908,A -85,B 0,C 180,E1 -9565.525,E2 -9565.525} C_VEL
LIN {X 0,Y 432.389,Z 148.251,A -85,B 0,C 180,E1 -9568.293,E2 -9568.293} C_VEL
LIN {X 0,Y 432.326,Z 148.26,A -85,B 0,C 180,E1 -9571.346,E2 -9571.346} C_VEL
LIN {X 0,Y 432.344,Z 148.255,A -85,B 0,C 180,E1 -9574.677,E2 -9574.677} C_VEL
LIN {X 0,Y 432.336,Z 148.254,A -85,B 0,C 180,E1 -9578.15,E2 -9578.15} C_VEL
LIN {X 0,Y 432.329,Z 148.258,A -85,B 0,C 180,E1 -9581.6,E2 -9581.6} C_VEL
LIN {X 0,Y 432.338,Z 148.25,A -85,B 0,C 180,E1 -9584.347,E2 -9584.347} C_VEL
LIN {X 0,Y 432.325,Z 148.255,A -85,B 0,C 180,E1 -9587.015,E2 -9587.015} C_VEL
LIN {X 0,Y 432.338,Z 148.251,A -85,B 0,C 180,E1 -9589.82,E2 -9589.82} C_VEL
LIN {X 0,Y 432.311,Z 148.261,A -85,B 0,C 180,E1 -9593.021,E2 -9593.021} C_VEL
LIN {X 0,Y 432.362,Z 148.255,A -85,B 0,C 180,E1 -9595.996,E2 -9595.996} C_VEL
LIN {X 0,Y 432.352,Z 148.256,A -85,B 0,C 180,E1 -9599.489,E2 -9599.489} C_VEL
LIN {X 0,Y 432.38,Z 148.344,A -85,B 0,C 180,E1 -9601.055,E2 -9601.055} C_VEL
LIN {X 0,Y 435.82,Z 160.775,A -85,B 0,C 180,E1 -9603.157,E2 -9603.157} C_VEL
LIN {X 0,Y 437.184,Z 165.922,A -85,B 0,C 180,E1 -9603.915,E2 -9603.915} C_VEL
LIN {X 0,Y 441.749,Z 176.844,A -85,B 0,C 180,E1 -9604.405,E2 -9604.405} C_VEL
LIN {X 0,Y 443.994,Z 186.642,A -85,B 0,C 180,E1 -9604.72,E2 -9604.72} C_VEL
LIN {X 0,Y 443.038,Z 251.933,A -85,B 0,C 180,E1 -9605.811,E2 -9605.811} C_VEL
LIN {X 0,Y 442.475,Z 257.778,A -85,B 0,C 180,E1 -9605.88,E2 -9605.88} C_VEL
LIN {X 0,Y 439.703,Z 267.3,A -85,B 0,C 180,E1 -9605.882,E2 -9605.882} C_VEL
LIN {X 0,Y 436.807,Z 276.827,A -85,B 0,C 180,E1 -9605.878,E2 -9605.878} C_VEL
LIN {X 0,Y 436.055,Z 282.687,A -85,B 0,C 180,E1 -9605.937,E2 -9605.937} C_VEL
LIN {X 0,Y 435.168,Z 334.032,A -85,B 0,C 180,E1 -9606.83,E2 -9606.83} C_VEL
LIN {X 0,Y 434.78,Z 349.022,A -85,B 0,C 180,E1 -9607.277,E2 -9607.277} C_VEL
LIN {X 0,Y 434.173,Z 363.151,A -85,B 0,C 180,E1 -9607.875,E2 -9607.875} C_VEL
LIN {X 0,Y 433.488,Z 376.334,A -85,B 0,C 180,E1 -9608.605,E2 -9608.605} C_VEL
LIN {X 0,Y 432.457,Z 390.017,A -85,B 0,C 180,E1 -9609.548,E2 -9609.548} C_VEL
LIN {X 0,Y 431.365,Z 402.541,A -85,B 0,C 180,E1 -9610.611,E2 -9610.611} C_VEL
LIN {X 0,Y 430.355,Z 413.88,A -85,B 0,C 180,E1 -9611.771,E2 -9611.771} C_VEL
LIN {X 0,Y 429.294,Z 424.853,A -85,B 0,C 180,E1 -9613.106,E2 -9613.106} C_VEL
LIN {X 0,Y 428.271,Z 434.722,A -85,B 0,C 180,E1 -9614.533,E2 -9614.533} C_VEL
LIN {X 0,Y 427.223,Z 444.647,A -85,B 0,C 180,E1 -9616.257,E2 -9616.257} C_VEL
LIN {X 0,Y 426.379,Z 453.351,A -85,B 0,C 180,E1 -9618.109,E2 -9618.109} C_VEL
LIN {X 0,Y 425.669,Z 460.601,A -85,B 0,C 180,E1 -9620.016,E2 -9620.016} C_VEL
LIN {X 0,Y 425.173,Z 466.344,A -85,B 0,C 180,E1 -9621.922,E2 -9621.922} C_VEL
LIN {X 0,Y 424.889,Z 469.732,A -85,B 0,C 180,E1 -9623.35,E2 -9623.35} C_VEL
LIN {X 0,Y 424.728,Z 473.179,A -85,B 0,C 180,E1 -9625.253,E2 -9625.253} C_VEL
LIN {X 0,Y 424.559,Z 475.459,A -85,B 0,C 180,E1 -9627.152,E2 -9627.152} C_VEL
LIN {X 0,Y 424.301,Z 476.634,A -85,B 0,C 180,E1 -9629.05,E2 -9629.05} C_VEL
LIN {X 0,Y 424.301,Z 476.649,A -85,B 0,C 180,E1 -9630.948,E2 -9630.948} C_VEL
LIN {X 0,Y 424.558,Z 475.534,A -85,B 0,C 180,E1 -9632.845,E2 -9632.845} C_VEL
LIN {X 0,Y 424.718,Z 473.318,A -85,B 0,C 180,E1 -9634.745,E2 -9634.745} C_VEL
LIN {X 0,Y 424.87,Z 469.944,A -85,B 0,C 180,E1 -9636.648,E2 -9636.648} C_VEL
LIN {X 0,Y 425.279,Z 465.3,A -85,B 0,C 180,E1 -9638.552,E2 -9638.552} C_VEL
LIN {X 0,Y 425.801,Z 459.273,A -85,B 0,C 180,E1 -9640.459,E2 -9640.459} C_VEL
LIN {X 0,Y 426.521,Z 451.681,A -85,B 0,C 180,E1 -9642.368,E2 -9642.368} C_VEL
LIN {X 0,Y 427.342,Z 443.786,A -85,B 0,C 180,E1 -9643.997,E2 -9643.997} C_VEL
LIN {X 0,Y 428.211,Z 435.323,A -85,B 0,C 180,E1 -9645.467,E2 -9645.467} C_VEL
LIN {X 0,Y 429.426,Z 423.77,A -85,B 0,C 180,E1 -9647.131,E2 -9647.131} C_VEL
LIN {X 0,Y 430.487,Z 412.305,A -85,B 0,C 180,E1 -9648.503,E2 -9648.503} C_VEL
LIN {X 0,Y 431.637,Z 399.741,A -85,B 0,C 180,E1 -9649.745,E2 -9649.745} C_VEL
LIN {X 0,Y 432.773,Z 386.593,A -85,B 0,C 180,E1 -9650.807,E2 -9650.807} C_VEL
LIN {X 0,Y 433.663,Z 373.06,A -85,B 0,C 180,E1 -9651.696,E2 -9651.696} C_VEL
LIN {X 0,Y 434.417,Z 357.869,A -85,B 0,C 180,E1 -9652.471,E2 -9652.471} C_VEL
LIN {X 0,Y 434.973,Z 343.218,A -85,B 0,C 180,E1 -9653.018,E2 -9653.018} C_VEL
LIN {X 0,Y 435.345,Z 328.492,A -85,B 0,C 180,E1 -9653.385,E2 -9653.385} C_VEL
LIN {X 0,Y 437.627,Z 187.995,A -85,B 0,C 180,E1 -9655.756,E2 -9655.756} C_VEL
LIN {X 0,Y 435.239,Z 178.194,A -85,B 0,C 180,E1 -9656.088,E2 -9656.088} C_VEL
LIN {X 0,Y 430,Z 165.999,A -85,B 0,C 180,E1 -9656.683,E2 -9656.683} C_VEL
LIN {X 0,Y 427.406,Z 156.406,A -85,B 0,C 180,E1 -9658.215,E2 -9658.215} C_VEL
LIN {X 0,Y 425.291,Z 149.137,A -85,B 0,C 180,E1 -9659.494,E2 -9659.494} C_VEL
LIN {X 0,Y 425.278,Z 149.133,A -85,B 0,C 180,E1 -9663.047,E2 -9663.047} C_VEL
LIN {X 0,Y 425.28,Z 149.135,A -85,B 0,C 180,E1 -9665.928,E2 -9665.928} C_VEL
LIN {X 0,Y 425.284,Z 149.125,A -85,B 0,C 180,E1 -9669.041,E2 -9669.041} C_VEL
LIN {X 0,Y 425.278,Z 149.134,A -85,B 0,C 180,E1 -9672.651,E2 -9672.651} C_VEL
LIN {X 0,Y 425.254,Z 149.137,A -85,B 0,C 180,E1 -9676.043,E2 -9676.043} C_VEL
LIN {X 0,Y 425.297,Z 149.13,A -85,B 0,C 180,E1 -9678.624,E2 -9678.624} C_VEL
LIN {X 0,Y 425.316,Z 149.126,A -85,B 0,C 180,E1 -9681.103,E2 -9681.103} C_VEL
LIN {X 0,Y 425.292,Z 149.132,A -85,B 0,C 180,E1 -9684.663,E2 -9684.663} C_VEL
LIN {X 0,Y 425.265,Z 149.134,A -85,B 0,C 180,E1 -9688.073,E2 -9688.073} C_VEL
LIN {X 0,Y 425.328,Z 149.128,A -85,B 0,C 180,E1 -9691.368,E2 -9691.368} C_VEL
LIN {X 0,Y 425.286,Z 149.129,A -85,B 0,C 180,E1 -9694.554,E2 -9694.554} C_VEL
LIN {X 0,Y 425.277,Z 149.134,A -85,B 0,C 180,E1 -9697.661,E2 -9697.661} C_VEL
LIN {X 0,Y 425.351,Z 149.116,A -85,B 0,C 180,E1 -9700.703,E2 -9700.703} C_VEL
LIN {X 0,Y 425.377,Z 149.121,A -85,B 0,C 180,E1 -9703.688,E2 -9703.688} C_VEL
LIN {X 0,Y 425.383,Z 149.11,A -85,B 0,C 180,E1 -9707.095,E2 -9707.095} C_VEL
LIN {X 0,Y 425.391,Z 149.122,A -85,B 0,C 180,E1 -9710.49,E2 -9710.49} C_VEL
LIN {X 0,Y 425.52,Z 149.089,A -85,B 0,C 180,E1 -9713.361,E2 -9713.361} C_VEL
LIN {X 0,Y 425.361,Z 149.123,A -85,B 0,C 180,E1 -9715.261,E2 -9715.261} C_VEL
LIN {X 0,Y 425.565,Z 149.097,A -85,B 0,C 180,E1 -9718.107,E2 -9718.107} C_VEL
LIN {X 0,Y 425.693,Z 149.069,A -85,B 0,C 180,E1 -9720,E2 -9720} C_VEL
LIN {X 0,Y 425.547,Z 149.103,A -85,B 0,C 180,E1 -9722.84,E2 -9722.84} C_VEL
LIN {X 0,Y 425.52,Z 149.091,A -85,B 0,C 180,E1 -9726.639,E2 -9726.639} C_VEL
LIN {X 0,Y 425.391,Z 149.116,A -85,B 0,C 180,E1 -9729.509,E2 -9729.509} C_VEL
LIN {X 0,Y 425.382,Z 149.106,A -85,B 0,C 180,E1 -9732.904,E2 -9732.904} C_VEL
LIN {X 0,Y 425.359,Z 149.123,A -85,B 0,C 180,E1 -9736.609,E2 -9736.609} C_VEL
LIN {X 0,Y 425.318,Z 149.116,A -85,B 0,C 180,E1 -9739.636,E2 -9739.636} C_VEL
LIN {X 0,Y 425.278,Z 149.136,A -85,B 0,C 180,E1 -9742.339,E2 -9742.339} C_VEL
LIN {X 0,Y 425.285,Z 149.126,A -85,B 0,C 180,E1 -9745.446,E2 -9745.446} C_VEL
LIN {X 0,Y 425.321,Z 149.123,A -85,B 0,C 180,E1 -9748.633,E2 -9748.633} C_VEL
LIN {X 0,Y 425.255,Z 149.138,A -85,B 0,C 180,E1 -9751.928,E2 -9751.928} C_VEL
LIN {X 0,Y 425.291,Z 149.129,A -85,B 0,C 180,E1 -9755.337,E2 -9755.337} C_VEL
LIN {X 0,Y 425.304,Z 149.114,A -85,B 0,C 180,E1 -9758.898,E2 -9758.898} C_VEL
LIN {X 0,Y 425.281,Z 149.119,A -85,B 0,C 180,E1 -9761.959,E2 -9761.959} C_VEL
LIN {X 0,Y 425.305,Z 149.131,A -85,B 0,C 180,E1 -9765.28,E2 -9765.28} C_VEL
LIN {X 0,Y 425.302,Z 149.133,A -85,B 0,C 180,E1 -9768.627,E2 -9768.627} C_VEL
LIN {X 0,Y 425.315,Z 149.127,A -85,B 0,C 180,E1 -9771.105,E2 -9771.105} C_VEL
LIN {X 0,Y 425.311,Z 149.262,A -85,B 0,C 180,E1 -9773.745,E2 -9773.745} C_VEL
LIN {X 0,Y 431.349,Z 168.988,A -85,B 0,C 180,E1 -9776.618,E2 -9776.618} C_VEL
LIN {X 0,Y 435.263,Z 182.48,A -85,B 0,C 180,E1 -9778.485,E2 -9778.485} C_VEL
LIN {X 0,Y 432.564,Z 214.102,A -85,B 0,C 180,E1 -9782.023,E2 -9782.023} C_VEL
LIN {X 0,Y 431.414,Z 229.321,A -85,B 0,C 180,E1 -9783.704,E2 -9783.704} C_VEL
LIN {X 0,Y 435.877,Z 265.107,A -85,B 0,C 180,E1 -9784.627,E2 -9784.627} C_VEL
LIN {X 0,Y 434.233,Z 375.764,A -85,B 0,C 180,E1 -9786.482,E2 -9786.482} C_VEL
LIN {X 0,Y 433.732,Z 402.422,A -85,B 0,C 180,E1 -9786.959,E2 -9786.959} C_VEL
LIN {X 0,Y 433.019,Z 418.074,A -85,B 0,C 180,E1 -9787.423,E2 -9787.423} C_VEL
LIN {X 0,Y 432.057,Z 432.492,A -85,B 0,C 180,E1 -9788.031,E2 -9788.031} C_VEL
LIN {X 0,Y 430.995,Z 447.281,A -85,B 0,C 180,E1 -9788.866,E2 -9788.866} C_VEL
LIN {X 0,Y 429.833,Z 460.416,A -85,B 0,C 180,E1 -9789.795,E2 -9789.795} C_VEL
LIN {X 0,Y 428.689,Z 473.984,A -85,B 0,C 180,E1 -9790.985,E2 -9790.985} C_VEL
LIN {X 0,Y 427.632,Z 486.05,A -85,B 0,C 180,E1 -9792.267,E2 -9792.267} C_VEL
LIN {X 0,Y 426.596,Z 497.583,A -85,B 0,C 180,E1 -9793.737,E2 -9793.737} C_VEL
LIN {X 0,Y 425.686,Z 508.52,A -85,B 0,C 180,E1 -9795.419,E2 -9795.419} C_VEL
LIN {X 0,Y 425.085,Z 517.519,A -85,B 0,C 180,E1 -9797.081,E2 -9797.081} C_VEL
LIN {X 0,Y 424.707,Z 524.18,A -85,B 0,C 180,E1 -9798.548,E2 -9798.548} C_VEL
LIN {X 0,Y 424.419,Z 531.44,A -85,B 0,C 180,E1 -9800.47,E2 -9800.47} C_VEL
LIN {X 0,Y 424.394,Z 537.163,A -85,B 0,C 180,E1 -9802.388,E2 -9802.388} C_VEL
LIN {X 0,Y 424.43,Z 541.485,A -85,B 0,C 180,E1 -9804.299,E2 -9804.299} C_VEL
LIN {X 0,Y 424.505,Z 544.518,A -85,B 0,C 180,E1 -9806.204,E2 -9806.204} C_VEL
LIN {X 0,Y 424.471,Z 546.322,A -85,B 0,C 180,E1 -9808.104,E2 -9808.104} C_VEL
LIN {X 0,Y 424.494,Z 546.94,A -85,B 0,C 180,E1 -9810.001,E2 -9810.001} C_VEL
LIN {X 0,Y 424.471,Z 546.322,A -85,B 0,C 180,E1 -9811.899,E2 -9811.899} C_VEL
LIN {X 0,Y 424.504,Z 544.517,A -85,B 0,C 180,E1 -9813.798,E2 -9813.798} C_VEL
LIN {X 0,Y 424.43,Z 541.476,A -85,B 0,C 180,E1 -9815.703,E2 -9815.703} C_VEL
LIN {X 0,Y 424.411,Z 537.145,A -85,B 0,C 180,E1 -9817.614,E2 -9817.614} C_VEL
LIN {X 0,Y 424.491,Z 531.425,A -85,B 0,C 180,E1 -9819.531,E2 -9819.531} C_VEL
LIN {X 0,Y 424.733,Z 524.162,A -85,B 0,C 180,E1 -9821.454,E2 -9821.454} C_VEL
LIN {X 0,Y 425.174,Z 516.318,A -85,B 0,C 180,E1 -9823.152,E2 -9823.152} C_VEL
LIN {X 0,Y 425.801,Z 507.035,A -85,B 0,C 180,E1 -9824.824,E2 -9824.824} C_VEL
LIN {X 0,Y 426.633,Z 497.538,A -85,B 0,C 180,E1 -9826.264,E2 -9826.264} C_VEL
LIN {X 0,Y 427.603,Z 485.676,A -85,B 0,C 180,E1 -9827.773,E2 -9827.773} C_VEL
LIN {X 0,Y 428.739,Z 472.643,A -85,B 0,C 180,E1 -9829.139,E2 -9829.139} C_VEL
LIN {X 0,Y 430.002,Z 458.758,A -85,B 0,C 180,E1 -9830.324,E2 -9830.324} C_VEL
LIN {X 0,Y 431.175,Z 445.351,A -85,B 0,C 180,E1 -9831.248,E2 -9831.248} C_VEL
LIN {X 0,Y 432.157,Z 431.357,A -85,B 0,C 180,E1 -9832.017,E2 -9832.017} C_VEL
LIN {X 0,Y 433.125,Z 416.028,A -85,B 0,C 180,E1 -9832.643,E2 -9832.643} C_VEL
LIN {X 0,Y 433.819,Z 400.774,A -85,B 0,C 180,E1 -9833.07,E2 -9833.07} C_VEL
LIN {X 0,Y 435.568,Z 289.575,A -85,B 0,C 180,E1 -9834.952,E2 -9834.952} C_VEL
LIN {X 0,Y 435.974,Z 270.155,A -85,B 0,C 180,E1 -9835.309,E2 -9835.309} C_VEL
LIN {X 0,Y 435.969,Z 263.407,A -85,B 0,C 180,E1 -9835.479,E2 -9835.479} C_VEL
LIN {X 0,Y 433.792,Z 242.129,A -85,B 0,C 180,E1 -9836.187,E2 -9836.187} C_VEL
LIN {X 0,Y 432.82,Z 235.212,A -85,B 0,C 180,E1 -9836.464,E2 -9836.464} C_VEL
LIN {X 0,Y 436.024,Z 208.218,A -85,B 0,C 180,E1 -9839.758,E2 -9839.758} C_VEL
LIN {X 0,Y 438.936,Z 189.665,A -85,B 0,C 180,E1 -9842.167,E2 -9842.167} C_VEL
LIN {X 0,Y 439.023,Z 187.876,A -85,B 0,C 180,E1 -9842.432,E2 -9842.432} C_VEL
LIN {X 0,Y 436.567,Z 178.452,A -85,B 0,C 180,E1 -9844.295,E2 -9844.295} C_VEL
LIN {X 0,Y 434.208,Z 171.304,A -85,B 0,C 180,E1 -9845.974,E2 -9845.974} C_VEL
LIN {X 0,Y 431.695,Z 164.626,A -85,B 0,C 180,E1 -9847.855,E2 -9847.855} C_VEL
LIN {X 0,Y 429.512,Z 159.3,A -85,B 0,C 180,E1 -9849.732,E2 -9849.732} C_VEL
LIN {X 0,Y 427.725,Z 155.194,A -85,B 0,C 180,E1 -9851.596,E2 -9851.596} C_VEL
LIN {X 0,Y 427.165,Z 153.659,A -85,B 0,C 180,E1 -9852.421,E2 -9852.421} C_VEL
LIN {X 0,Y 425.72,Z 150.852,A -85,B 0,C 180,E1 -9854.776,E2 -9854.776} C_VEL
LIN {X 0,Y 425.337,Z 149.634,A -85,B 0,C 180,E1 -9856.639,E2 -9856.639} C_VEL
LIN {X 0,Y 425.322,Z 149.564,A -85,B 0,C 180,E1 -9858.627,E2 -9858.627} C_VEL
LIN {X 0,Y 425.845,Z 151.206,A -85,B 0,C 180,E1 -9861.161,E2 -9861.161} C_VEL
LIN {X 0,Y 426.595,Z 152.49,A -85,B 0,C 180,E1 -9862.442,E2 -9862.442} C_VEL
LIN {X 0,Y 428.277,Z 156.822,A -85,B 0,C 180,E1 -9865.136,E2 -9865.136} C_VEL
LIN {X 0,Y 430.016,Z 161.674,A -85,B 0,C 180,E1 -9867.362,E2 -9867.362} C_VEL
LIN {X 0,Y 432.197,Z 168.901,A -85,B 0,C 180,E1 -9870,E2 -9870} C_VEL
LIN {X 0,Y 434.294,Z 177.161,A -85,B 0,C 180,E1 -9872.536,E2 -9872.536} C_VEL
LIN {X 0,Y 435.441,Z 183.184,A -85,B 0,C 180,E1 -9874.165,E2 -9874.165} C_VEL
LIN {X 0,Y 435.301,Z 186.812,A -85,B 0,C 180,E1 -9874.993,E2 -9874.993} C_VEL
LIN {X 0,Y 433.116,Z 203.09,A -85,B 0,C 180,E1 -9878.337,E2 -9878.337} C_VEL
LIN {X 0,Y 432.711,Z 207.244,A -85,B 0,C 180,E1 -9879.131,E2 -9879.131} C_VEL
LIN {X 0,Y 436.655,Z 222.638,A -85,B 0,C 180,E1 -9879.986,E2 -9879.986} C_VEL
LIN {X 0,Y 433.257,Z 291.383,A -85,B 0,C 180,E1 -9881.866,E2 -9881.866} C_VEL
LIN {X 0,Y 432.078,Z 325.203,A -85,B 0,C 180,E1 -9882.793,E2 -9882.793} C_VEL
LIN {X 0,Y 431.683,Z 339.426,A -85,B 0,C 180,E1 -9883.386,E2 -9883.386} C_VEL
LIN {X 0,Y 431.164,Z 352.48,A -85,B 0,C 180,E1 -9884.132,E2 -9884.132} C_VEL
LIN {X 0,Y 430.479,Z 364.148,A -85,B 0,C 180,E1 -9884.979,E2 -9884.979} C_VEL
LIN {X 0,Y 429.749,Z 375.811,A -85,B 0,C 180,E1 -9886.042,E2 -9886.042} C_VEL
LIN {X 0,Y 429.014,Z 386.215,A -85,B 0,C 180,E1 -9887.223,E2 -9887.223} C_VEL
LIN {X 0,Y 428.387,Z 394.754,A -85,B 0,C 180,E1 -9888.406,E2 -9888.406} C_VEL
LIN {X 0,Y 427.688,Z 403.166,A -85,B 0,C 180,E1 -9889.825,E2 -9889.825} C_VEL
LIN {X 0,Y 426.995,Z 410.098,A -85,B 0,C 180,E1 -9891.294,E2 -9891.294} C_VEL
LIN {X 0,Y 426.528,Z 415.986,A -85,B 0,C 180,E1 -9892.901,E2 -9892.901} C_VEL
LIN {X 0,Y 426.026,Z 419.976,A -85,B 0,C 180,E1 -9894.32,E2 -9894.32} C_VEL
LIN {X 0,Y 425.858,Z 422.031,A -85,B 0,C 180,E1 -9895.267,E2 -9895.267} C_VEL
LIN {X 0,Y 425.76,Z 423.588,A -85,B 0,C 180,E1 -9896.214,E2 -9896.214} C_VEL
LIN {X 0,Y 425.594,Z 424.727,A -85,B 0,C 180,E1 -9897.16,E2 -9897.16} C_VEL
LIN {X 0,Y 425.481,Z 425.458,A -85,B 0,C 180,E1 -9898.107,E2 -9898.107} C_VEL
LIN {X 0,Y 425.364,Z 425.784,A -85,B 0,C 180,E1 -9899.053,E2 -9899.053} C_VEL
LIN {X 0,Y 425.301,Z 425.649,A -85,B 0,C 180,E1 -9900,E2 -9900} C_VEL
LIN {X 0,Y 425.317,Z 425.094,A -85,B 0,C 180,E1 -9900.947,E2 -9900.947} C_VEL
LIN {X 0,Y 425.235,Z 424.154,A -85,B 0,C 180,E1 -9901.894,E2 -9901.894} C_VEL
LIN {X 0,Y 425.352,Z 422.776,A -85,B 0,C 180,E1 -9902.841,E2 -9902.841} C_VEL
LIN {X 0,Y 425.303,Z 419.898,A -85,B 0,C 180,E1 -9904.265,E2 -9904.265} C_VEL
LIN {X 0,Y 425.537,Z 415.953,A -85,B 0,C 180,E1 -9905.687,E2 -9905.687} C_VEL
LIN {X 0,Y 425.83,Z 410.872,A -85,B 0,C 180,E1 -9907.111,E2 -9907.111} C_VEL
LIN {X 0,Y 426.022,Z 404.504,A -85,B 0,C 180,E1 -9908.538,E2 -9908.538} C_VEL
LIN {X 0,Y 426.465,Z 396.603,A -85,B 0,C 180,E1 -9909.965,E2 -9909.965} C_VEL
LIN {X 0,Y 426.89,Z 386.875,A -85,B 0,C 180,E1 -9911.394,E2 -9911.394} C_VEL
LIN {X 0,Y 427.358,Z 376.824,A -85,B 0,C 180,E1 -9912.586,E2 -9912.586} C_VEL
LIN {X 0,Y 427.895,Z 365.768,A -85,B 0,C 180,E1 -9913.657,E2 -9913.657} C_VEL
LIN {X 0,Y 428.318,Z 353.56,A -85,B 0,C 180,E1 -9914.612,E2 -9914.612} C_VEL
LIN {X 0,Y 428.776,Z 339.619,A -85,B 0,C 180,E1 -9915.447,E2 -9915.447} C_VEL
LIN {X 0,Y 429.067,Z 326.939,A -85,B 0,C 180,E1 -9916.016,E2 -9916.016} C_VEL
LIN {X 0,Y 429.355,Z 313.199,A -85,B 0,C 180,E1 -9916.432,E2 -9916.432} C_VEL
LIN {X 0,Y 431.059,Z 217.536,A -85,B 0,C 180,E1 -9918.432,E2 -9918.432} C_VEL
LIN {X 0,Y 428.009,Z 200.188,A -85,B 0,C 180,E1 -9918.967,E2 -9918.967} C_VEL
LIN {X 0,Y 428.938,Z 182.405,A -85,B 0,C 180,E1 -9922.139,E2 -9922.139} C_VEL
LIN {X 0,Y 429.698,Z 169.921,A -85,B 0,C 180,E1 -9924.392,E2 -9924.392} C_VEL
LIN {X 0,Y 427.81,Z 160.129,A -85,B 0,C 180,E1 -9926.331,E2 -9926.331} C_VEL
LIN {X 0,Y 425.321,Z 149.131,A -85,B 0,C 180,E1 -9928.599,E2 -9928.599} C_VEL
LIN {X 0,Y 425.27,Z 149.137,A -85,B 0,C 180,E1 -9931.927,E2 -9931.927} C_VEL
LIN {X 0,Y 425.304,Z 149.136,A -85,B 0,C 180,E1 -9935.336,E2 -9935.336} C_VEL
LIN {X 0,Y 425.296,Z 149.133,A -85,B 0,C 180,E1 -9938.899,E2 -9938.899} C_VEL
LIN {X 0,Y 425.287,Z 149.133,A -85,B 0,C 180,E1 -9941.957,E2 -9941.957} C_VEL
LIN {X 0,Y 425.29,Z 149.136,A -85,B 0,C 180,E1 -9945.283,E2 -9945.283} C_VEL
LIN {X 0,Y 425.279,Z 149.137,A -85,B 0,C 180,E1 -9948.621,E2 -9948.621} C_VEL
LIN {X 0,Y 425.303,Z 149.137,A -85,B 0,C 180,E1 -9951.101,E2 -9951.101} C_VEL
LIN {X 0,Y 425.303,Z 149.135,A -85,B 0,C 180,E1 -9954.663,E2 -9954.663} C_VEL
LIN {X 0,Y 425.269,Z 149.139,A -85,B 0,C 180,E1 -9958.072,E2 -9958.072} C_VEL
LIN {X 0,Y 425.314,Z 149.3,A -85,B 0,C 180,E1 -9960.627,E2 -9960.627} C_VEL
LIN {X 0,Y 428.743,Z 161.256,A -85,B 0,C 180,E1 -9962.678,E2 -9962.678} C_VEL
LIN {X 0,Y 430.1,Z 166.304,A -85,B 0,C 180,E1 -9963.449,E2 -9963.449} C_VEL
LIN {X 0,Y 435.833,Z 179.955,A -85,B 0,C 180,E1 -9964.08,E2 -9964.08} C_VEL
LIN {X 0,Y 437.555,Z 187.419,A -85,B 0,C 180,E1 -9964.326,E2 -9964.326} C_VEL
LIN {X 0,Y 436.055,Z 282.687,A -85,B 0,C 180,E1 -9965.937,E2 -9965.937} C_VEL
LIN {X 0,Y 435.354,Z 288.531,A -85,B 0,C 180,E1 -9965.999,E2 -9965.999} C_VEL
LIN {X 0,Y 429.851,Z 307.578,A -85,B 0,C 180,E1 -9966.009,E2 -9966.009} C_VEL
LIN {X 0,Y 429.101,Z 313.424,A -85,B 0,C 180,E1 -9966.069,E2 -9966.069} C_VEL
LIN {X 0,Y 428.644,Z 336.037,A -85,B 0,C 180,E1 -9966.491,E2 -9966.491} C_VEL
LIN {X 0,Y 428.158,Z 351.75,A -85,B 0,C 180,E1 -9966.987,E2 -9966.987} C_VEL
LIN {X 0,Y 427.491,Z 366.881,A -85,B 0,C 180,E1 -9967.676,E2 -9967.676} C_VEL
LIN {X 0,Y 426.645,Z 380.706,A -85,B 0,C 180,E1 -9968.498,E2 -9968.498} C_VEL
LIN {X 0,Y 425.587,Z 393.635,A -85,B 0,C 180,E1 -9969.456,E2 -9969.456} C_VEL
LIN {X 0,Y 424.502,Z 405.607,A -85,B 0,C 180,E1 -9970.537,E2 -9970.537} C_VEL
LIN {X 0,Y 423.395,Z 416.77,A -85,B 0,C 180,E1 -9971.74,E2 -9971.74} C_VEL
LIN {X 0,Y 422.305,Z 427.16,A -85,B 0,C 180,E1 -9973.067,E2 -9973.067} C_VEL
LIN {X 0,Y 421.28,Z 436.762,A -85,B 0,C 180,E1 -9974.518,E2 -9974.518} C_VEL
LIN {X 0,Y 420.307,Z 445.493,A -85,B 0,C 180,E1 -9976.08,E2 -9976.08} C_VEL
LIN {X 0,Y 419.454,Z 453.935,A -85,B 0,C 180,E1 -9977.909,E2 -9977.909} C_VEL
LIN {X 0,Y 418.696,Z 461.186,A -85,B 0,C 180,E1 -9979.848,E2 -9979.848} C_VEL
LIN {X 0,Y 418.17,Z 466.929,A -85,B 0,C 180,E1 -9981.786,E2 -9981.786} C_VEL
LIN {X 0,Y 417.867,Z 470.317,A -85,B 0,C 180,E1 -9983.238,E2 -9983.238} C_VEL
LIN {X 0,Y 417.685,Z 473.763,A -85,B 0,C 180,E1 -9985.173,E2 -9985.173} C_VEL
LIN {X 0,Y 417.515,Z 476.043,A -85,B 0,C 180,E1 -9987.104,E2 -9987.104} C_VEL
LIN {X 0,Y 417.244,Z 477.218,A -85,B 0,C 180,E1 -9989.034,E2 -9989.034} C_VEL
LIN {X 0,Y 417.243,Z 477.232,A -85,B 0,C 180,E1 -9990.964,E2 -9990.964} C_VEL
LIN {X 0,Y 417.514,Z 476.116,A -85,B 0,C 180,E1 -9992.893,E2 -9992.893} C_VEL
LIN {X 0,Y 417.674,Z 473.901,A -85,B 0,C 180,E1 -9994.825,E2 -9994.825} C_VEL
LIN {X 0,Y 417.85,Z 470.526,A -85,B 0,C 180,E1 -9996.76,E2 -9996.76} C_VEL
LIN {X 0,Y 418.258,Z 465.885,A -85,B 0,C 180,E1 -9998.697,E2 -9998.697} C_VEL
LIN {X 0,Y 418.842,Z 459.854,A -85,B 0,C 180,E1 -10000.635,E2 -10000.635} C_VEL
LIN {X 0,Y 419.598,Z 452.262,A -85,B 0,C 180,E1 -10002.575,E2 -10002.575} C_VEL
LIN {X 0,Y 420.416,Z 444.701,A -85,B 0,C 180,E1 -10004.17,E2 -10004.17} C_VEL
LIN {X 0,Y 421.394,Z 435.899,A -85,B 0,C 180,E1 -10005.723,E2 -10005.723} C_VEL
LIN {X 0,Y 422.443,Z 426.123,A -85,B 0,C 180,E1 -10007.174,E2 -10007.174} C_VEL
LIN {X 0,Y 423.685,Z 414.183,A -85,B 0,C 180,E1 -10008.658,E2 -10008.658} C_VEL
LIN {X 0,Y 424.875,Z 401.616,A -85,B 0,C 180,E1 -10009.946,E2 -10009.946} C_VEL
LIN {X 0,Y 426.032,Z 388.738,A -85,B 0,C 180,E1 -10011.025,E2 -10011.025} C_VEL
LIN {X 0,Y 427.013,Z 374.597,A -85,B 0,C 180,E1 -10011.988,E2 -10011.988} C_VEL
LIN {X 0,Y 427.813,Z 361.2,A -85,B 0,C 180,E1 -10012.7,E2 -10012.7} C_VEL
LIN {X 0,Y 428.391,Z 345.942,A -85,B 0,C 180,E1 -10013.315,E2 -10013.315} C_VEL
LIN {X 0,Y 428.805,Z 330.513,A -85,B 0,C 180,E1 -10013.728,E2 -10013.728} C_VEL
LIN {X 0,Y 431.246,Z 189.195,A -85,B 0,C 180,E1 -10016.152,E2 -10016.152} C_VEL
LIN {X 0,Y 429.162,Z 180.805,A -85,B 0,C 180,E1 -10016.446,E2 -10016.446} C_VEL
LIN {X 0,Y 422.982,Z 166.583,A -85,B 0,C 180,E1 -10017.154,E2 -10017.154} C_VEL
LIN {X 0,Y 419.707,Z 154.992,A -85,B 0,C 180,E1 -10019.05,E2 -10019.05} C_VEL
LIN {X 0,Y 418.238,Z 150.014,A -85,B 0,C 180,E1 -10019.958,E2 -10019.958} C_VEL
LIN {X 0,Y 418.244,Z 150.017,A -85,B 0,C 180,E1 -10023.676,E2 -10023.676} C_VEL
LIN {X 0,Y 418.24,Z 150.012,A -85,B 0,C 180,E1 -10027.222,E2 -10027.222} C_VEL
LIN {X 0,Y 418.241,Z 149.993,A -85,B 0,C 180,E1 -10029.681,E2 -10029.681} C_VEL
LIN {X 0,Y 418.239,Z 150.011,A -85,B 0,C 180,E1 -10032.322,E2 -10032.322} C_VEL
LIN {X 0,Y 418.231,Z 150.01,A -85,B 0,C 180,E1 -10035.108,E2 -10035.108} C_VEL
LIN {X 0,Y 418.249,Z 150.007,A -85,B 0,C 180,E1 -10037.768,E2 -10037.768} C_VEL
LIN {X 0,Y 418.261,Z 150.007,A -85,B 0,C 180,E1 -10040.615,E2 -10040.615} C_VEL
LIN {X 0,Y 418.238,Z 150.009,A -85,B 0,C 180,E1 -10043.975,E2 -10043.975} C_VEL
LIN {X 0,Y 418.252,Z 150.012,A -85,B 0,C 180,E1 -10047.154,E2 -10047.154} C_VEL
LIN {X 0,Y 418.265,Z 149.999,A -85,B 0,C 180,E1 -10050.838,E2 -10050.838} C_VEL
LIN {X 0,Y 418.261,Z 150.003,A -85,B 0,C 180,E1 -10054.095,E2 -10054.095} C_VEL
LIN {X 0,Y 418.222,Z 150.016,A -85,B 0,C 180,E1 -10057.263,E2 -10057.263} C_VEL
LIN {X 0,Y 418.273,Z 149.999,A -85,B 0,C 180,E1 -10060.364,E2 -10060.364} C_VEL
LIN {X 0,Y 418.306,Z 150.003,A -85,B 0,C 180,E1 -10063.404,E2 -10063.404} C_VEL
LIN {X 0,Y 418.336,Z 149.987,A -85,B 0,C 180,E1 -10066.998,E2 -10066.998} C_VEL
LIN {X 0,Y 418.331,Z 150,A -85,B 0,C 180,E1 -10070.328,E2 -10070.328} C_VEL
LIN {X 0,Y 418.482,Z 149.966,A -85,B 0,C 180,E1 -10073.249,E2 -10073.249} C_VEL
LIN {X 0,Y 418.331,Z 149.999,A -85,B 0,C 180,E1 -10075.181,E2 -10075.181} C_VEL
LIN {X 0,Y 418.534,Z 149.973,A -85,B 0,C 180,E1 -10078.075,E2 -10078.075} C_VEL
LIN {X 0,Y 418.663,Z 149.944,A -85,B 0,C 180,E1 -10080,E2 -10080} C_VEL
LIN {X 0,Y 418.501,Z 149.98,A -85,B 0,C 180,E1 -10082.888,E2 -10082.888} C_VEL
LIN {X 0,Y 418.482,Z 149.966,A -85,B 0,C 180,E1 -10086.751,E2 -10086.751} C_VEL
LIN {X 0,Y 418.331,Z 149.995,A -85,B 0,C 180,E1 -10089.671,E2 -10089.671} C_VEL
LIN {X 0,Y 418.335,Z 149.983,A -85,B 0,C 180,E1 -10093.001,E2 -10093.001} C_VEL
LIN {X 0,Y 418.309,Z 149.999,A -85,B 0,C 180,E1 -10096.739,E2 -10096.739} C_VEL
LIN {X 0,Y 418.26,Z 149.996,A -85,B 0,C 180,E1 -10099.791,E2 -10099.791} C_VEL
LIN {X 0,Y 418.228,Z 150.009,A -85,B 0,C 180,E1 -10102.737,E2 -10102.737} C_VEL
LIN {X 0,Y 418.26,Z 150.003,A -85,B 0,C 180,E1 -10105.905,E2 -10105.905} C_VEL
LIN {X 0,Y 418.254,Z 149.999,A -85,B 0,C 180,E1 -10109.163,E2 -10109.163} C_VEL
LIN {X 0,Y 418.247,Z 150.007,A -85,B 0,C 180,E1 -10112.845,E2 -10112.845} C_VEL
LIN {X 0,Y 418.239,Z 150.016,A -85,B 0,C 180,E1 -10116.24,E2 -10116.24} C_VEL
LIN {X 0,Y 418.243,Z 149.984,A -85,B 0,C 180,E1 -10119.683,E2 -10119.683} C_VEL
LIN {X 0,Y 418.22,Z 150.004,A -85,B 0,C 180,E1 -10122.322,E2 -10122.322} C_VEL
LIN {X 0,Y 418.25,Z 150.009,A -85,B 0,C 180,E1 -10125.113,E2 -10125.113} C_VEL
LIN {X 0,Y 418.285,Z 150.008,A -85,B 0,C 180,E1 -10127.775,E2 -10127.775} C_VEL
LIN {X 0,Y 418.258,Z 150.009,A -85,B 0,C 180,E1 -10131.561,E2 -10131.561} C_VEL
LIN {X 0,Y 418.25,Z 150.198,A -85,B 0,C 180,E1 -10133.331,E2 -10133.331} C_VEL
LIN {X 0,Y 424.472,Z 170.456,A -85,B 0,C 180,E1 -10136.346,E2 -10136.346} C_VEL
LIN {X 0,Y 428.533,Z 184.751,A -85,B 0,C 180,E1 -10138.347,E2 -10138.347} C_VEL
LIN {X 0,Y 425.628,Z 216.271,A -85,B 0,C 180,E1 -10141.929,E2 -10141.929} C_VEL
LIN {X 0,Y 424.8,Z 228.29,A -85,B 0,C 180,E1 -10143.254,E2 -10143.254} C_VEL
LIN {X 0,Y 429.399,Z 265.211,A -85,B 0,C 180,E1 -10144.226,E2 -10144.226} C_VEL
LIN {X 0,Y 428.098,Z 353.728,A -85,B 0,C 180,E1 -10145.738,E2 -10145.738} C_VEL
LIN {X 0,Y 427.256,Z 400.701,A -85,B 0,C 180,E1 -10146.557,E2 -10146.557} C_VEL
LIN {X 0,Y 426.53,Z 415.945,A -85,B 0,C 180,E1 -10146.996,E2 -10146.996} C_VEL
LIN {X 0,Y 425.534,Z 430.742,A -85,B 0,C 180,E1 -10147.612,E2 -10147.612} C_VEL
LIN {X 0,Y 424.466,Z 445.316,A -85,B 0,C 180,E1 -10148.428,E2 -10148.428} C_VEL
LIN {X 0,Y 423.094,Z 459.842,A -85,B 0,C 180,E1 -10149.459,E2 -10149.459} C_VEL
LIN {X 0,Y 421.9,Z 473.405,A -85,B 0,C 180,E1 -10150.667,E2 -10150.667} C_VEL
LIN {X 0,Y 420.695,Z 485.977,A -85,B 0,C 180,E1 -10152.03,E2 -10152.03} C_VEL
LIN {X 0,Y 419.683,Z 496.996,A -85,B 0,C 180,E1 -10153.462,E2 -10153.462} C_VEL
LIN {X 0,Y 418.7,Z 507.93,A -85,B 0,C 180,E1 -10155.17,E2 -10155.17} C_VEL
LIN {X 0,Y 418.041,Z 517.267,A -85,B 0,C 180,E1 -10156.933,E2 -10156.933} C_VEL
LIN {X 0,Y 417.599,Z 525.573,A -85,B 0,C 180,E1 -10158.842,E2 -10158.842} C_VEL
LIN {X 0,Y 417.322,Z 532.429,A -85,B 0,C 180,E1 -10160.795,E2 -10160.795} C_VEL
LIN {X 0,Y 417.337,Z 537.807,A -85,B 0,C 180,E1 -10162.745,E2 -10162.745} C_VEL
LIN {X 0,Y 417.349,Z 540.898,A -85,B 0,C 180,E1 -10164.202,E2 -10164.202} C_VEL
LIN {X 0,Y 417.421,Z 543.932,A -85,B 0,C 180,E1 -10166.14,E2 -10166.14} C_VEL
LIN {X 0,Y 417.413,Z 545.738,A -85,B 0,C 180,E1 -10168.072,E2 -10168.072} C_VEL
LIN {X 0,Y 417.421,Z 546.355,A -85,B 0,C 180,E1 -10170.001,E2 -10170.001} C_VEL
LIN {X 0,Y 417.414,Z 545.738,A -85,B 0,C 180,E1 -10171.931,E2 -10171.931} C_VEL
LIN {X 0,Y 417.419,Z 543.93,A -85,B 0,C 180,E1 -10173.863,E2 -10173.863} C_VEL
LIN {X 0,Y 417.349,Z 540.888,A -85,B 0,C 180,E1 -10175.8,E2 -10175.8} C_VEL
LIN {X 0,Y 417.331,Z 536.555,A -85,B 0,C 180,E1 -10177.744,E2 -10177.744} C_VEL
LIN {X 0,Y 417.399,Z 530.831,A -85,B 0,C 180,E1 -10179.695,E2 -10179.695} C_VEL
LIN {X 0,Y 417.695,Z 523.569,A -85,B 0,C 180,E1 -10181.65,E2 -10181.65} C_VEL
LIN {X 0,Y 418.153,Z 515.921,A -85,B 0,C 180,E1 -10183.338,E2 -10183.338} C_VEL
LIN {X 0,Y 418.836,Z 506.443,A -85,B 0,C 180,E1 -10185.076,E2 -10185.076} C_VEL
LIN {X 0,Y 419.702,Z 496.946,A -85,B 0,C 180,E1 -10186.54,E2 -10186.54} C_VEL
LIN {X 0,Y 420.694,Z 485.564,A -85,B 0,C 180,E1 -10188.016,E2 -10188.016} C_VEL
LIN {X 0,Y 421.835,Z 473.311,A -85,B 0,C 180,E1 -10189.338,E2 -10189.338} C_VEL
LIN {X 0,Y 423.143,Z 459.746,A -85,B 0,C 180,E1 -10190.541,E2 -10190.541} C_VEL
LIN {X 0,Y 424.492,Z 445.085,A -85,B 0,C 180,E1 -10191.58,E2 -10191.58} C_VEL
LIN {X 0,Y 425.472,Z 431.768,A -85,B 0,C 180,E1 -10192.33,E2 -10192.33} C_VEL
LIN {X 0,Y 426.491,Z 416.522,A -85,B 0,C 180,E1 -10192.977,E2 -10192.977} C_VEL
LIN {X 0,Y 427.234,Z 401.582,A -85,B 0,C 180,E1 -10193.415,E2 -10193.415} C_VEL
LIN {X 0,Y 428.26,Z 345.981,A -85,B 0,C 180,E1 -10194.384,E2 -10194.384} C_VEL
LIN {X 0,Y 429.282,Z 284.466,A -85,B 0,C 180,E1 -10195.454,E2 -10195.454} C_VEL
LIN {X 0,Y 429.865,Z 264.808,A -85,B 0,C 180,E1 -10195.916,E2 -10195.916} C_VEL
LIN {X 0,Y 427.748,Z 243.234,A -85,B 0,C 180,E1 -10196.665,E2 -10196.665} C_VEL
LIN {X 0,Y 426.505,Z 234.86,A -85,B 0,C 180,E1 -10197.005,E2 -10197.005} C_VEL
LIN {X 0,Y 429.863,Z 209.313,A -85,B 0,C 180,E1 -10200.217,E2 -10200.217} C_VEL
LIN {X 0,Y 432.871,Z 191.112,A -85,B 0,C 180,E1 -10202.658,E2 -10202.658} C_VEL
LIN {X 0,Y 430.709,Z 182.281,A -85,B 0,C 180,E1 -10204.445,E2 -10204.445} C_VEL
LIN {X 0,Y 428.383,Z 175.057,A -85,B 0,C 180,E1 -10206.202,E2 -10206.202} C_VEL
LIN {X 0,Y 425.74,Z 167.74,A -85,B 0,C 180,E1 -10208.362,E2 -10208.362} C_VEL
LIN {X 0,Y 423.622,Z 162.621,A -85,B 0,C 180,E1 -10210.318,E2 -10210.318} C_VEL
LIN {X 0,Y 422.371,Z 159.759,A -85,B 0,C 180,E1 -10211.728,E2 -10211.728} C_VEL
LIN {X 0,Y 421.375,Z 157.464,A -85,B 0,C 180,E1 -10213.145,E2 -10213.145} C_VEL
LIN {X 0,Y 420.295,Z 155.155,A -85,B 0,C 180,E1 -10215.388,E2 -10215.388} C_VEL
LIN {X 0,Y 420.039,Z 154.214,A -85,B 0,C 180,E1 -10217.41,E2 -10217.41} C_VEL
LIN {X 0,Y 420.07,Z 154.547,A -85,B 0,C 180,E1 -10219.27,E2 -10219.27} C_VEL
LIN {X 0,Y 420.774,Z 156.439,A -85,B 0,C 180,E1 -10221.83,E2 -10221.83} C_VEL
LIN {X 0,Y 422.162,Z 159.869,A -85,B 0,C 180,E1 -10224.362,E2 -10224.362} C_VEL
LIN {X 0,Y 423.908,Z 164.696,A -85,B 0,C 180,E1 -10226.831,E2 -10226.831} C_VEL
LIN {X 0,Y 425.981,Z 171.693,A -85,B 0,C 180,E1 -10229.574,E2 -10229.574} C_VEL
LIN {X 0,Y 427.913,Z 179.502,A -85,B 0,C 180,E1 -10232.091,E2 -10232.091} C_VEL
LIN {X 0,Y 429,Z 185.359,A -85,B 0,C 180,E1 -10233.748,E2 -10233.748} C_VEL
LIN {X 0,Y 429.12,Z 188.768,A -85,B 0,C 180,E1 -10234.587,E2 -10234.587} C_VEL
LIN {X 0,Y 426.912,Z 203.776,A -85,B 0,C 180,E1 -10237.751,E2 -10237.751} C_VEL
LIN {X 0,Y 426.457,Z 207.854,A -85,B 0,C 180,E1 -10238.552,E2 -10238.552} C_VEL
LIN {X 0,Y 430.24,Z 222.512,A -85,B 0,C 180,E1 -10239.424,E2 -10239.424} C_VEL
LIN {X 0,Y 430.7,Z 225.009,A -85,B 0,C 180,E1 -10239.548,E2 -10239.548} C_VEL
LIN {X 0,Y 426.1,Z 312.146,A -85,B 0,C 180,E1 -10241.986,E2 -10241.986} C_VEL
LIN {X 0,Y 425.65,Z 328.575,A -85,B 0,C 180,E1 -10242.494,E2 -10242.494} C_VEL
LIN {X 0,Y 425.131,Z 342.544,A -85,B 0,C 180,E1 -10243.122,E2 -10243.122} C_VEL
LIN {X 0,Y 424.486,Z 355.798,A -85,B 0,C 180,E1 -10243.927,E2 -10243.927} C_VEL
LIN {X 0,Y 423.756,Z 367.777,A -85,B 0,C 180,E1 -10244.858,E2 -10244.858} C_VEL
LIN {X 0,Y 422.912,Z 379.975,A -85,B 0,C 180,E1 -10246.057,E2 -10246.057} C_VEL
LIN {X 0,Y 422.193,Z 389.816,A -85,B 0,C 180,E1 -10247.258,E2 -10247.258} C_VEL
LIN {X 0,Y 421.376,Z 399.347,A -85,B 0,C 180,E1 -10248.698,E2 -10248.698} C_VEL
LIN {X 0,Y 420.633,Z 407.06,A -85,B 0,C 180,E1 -10250.139,E2 -10250.139} C_VEL
LIN {X 0,Y 420.029,Z 412.287,A -85,B 0,C 180,E1 -10251.339,E2 -10251.339} C_VEL
LIN {X 0,Y 419.62,Z 417.344,A -85,B 0,C 180,E1 -10252.784,E2 -10252.784} C_VEL
LIN {X 0,Y 419.08,Z 421.265,A -85,B 0,C 180,E1 -10254.225,E2 -10254.225} C_VEL
LIN {X 0,Y 418.895,Z 423.273,A -85,B 0,C 180,E1 -10255.188,E2 -10255.188} C_VEL
LIN {X 0,Y 418.777,Z 424.78,A -85,B 0,C 180,E1 -10256.151,E2 -10256.151} C_VEL
LIN {X 0,Y 418.599,Z 425.889,A -85,B 0,C 180,E1 -10257.113,E2 -10257.113} C_VEL
LIN {X 0,Y 418.497,Z 426.581,A -85,B 0,C 180,E1 -10258.075,E2 -10258.075} C_VEL
LIN {X 0,Y 418.348,Z 426.861,A -85,B 0,C 180,E1 -10259.038,E2 -10259.038} C_VEL
LIN {X 0,Y 418.277,Z 426.678,A -85,B 0,C 180,E1 -10260,E2 -10260} C_VEL
LIN {X 0,Y 418.292,Z 426.082,A -85,B 0,C 180,E1 -10260.963,E2 -10260.963} C_VEL
LIN {X 0,Y 418.212,Z 425.104,A -85,B 0,C 180,E1 -10261.926,E2 -10261.926} C_VEL
LIN {X 0,Y 418.327,Z 423.667,A -85,B 0,C 180,E1 -10262.889,E2 -10262.889} C_VEL
LIN {X 0,Y 418.285,Z 420.716,A -85,B 0,C 180,E1 -10264.336,E2 -10264.336} C_VEL
LIN {X 0,Y 418.533,Z 416.687,A -85,B 0,C 180,E1 -10265.783,E2 -10265.783} C_VEL
LIN {X 0,Y 418.85,Z 410.515,A -85,B 0,C 180,E1 -10267.472,E2 -10267.472} C_VEL
LIN {X 0,Y 419.096,Z 403.82,A -85,B 0,C 180,E1 -10268.924,E2 -10268.924} C_VEL
LIN {X 0,Y 419.547,Z 395.554,A -85,B 0,C 180,E1 -10270.374,E2 -10270.374} C_VEL
LIN {X 0,Y 420.007,Z 385.248,A -85,B 0,C 180,E1 -10271.828,E2 -10271.828} C_VEL
LIN {X 0,Y 420.542,Z 374.684,A -85,B 0,C 180,E1 -10273.039,E2 -10273.039} C_VEL
LIN {X 0,Y 421.131,Z 363.011,A -85,B 0,C 180,E1 -10274.114,E2 -10274.114} C_VEL
LIN {X 0,Y 421.483,Z 351.444,A -85,B 0,C 180,E1 -10274.978,E2 -10274.978} C_VEL
LIN {X 0,Y 421.931,Z 339.049,A -85,B 0,C 180,E1 -10275.704,E2 -10275.704} C_VEL
LIN {X 0,Y 422.203,Z 326.628,A -85,B 0,C 180,E1 -10276.252,E2 -10276.252} C_VEL
LIN {X 0,Y 422.472,Z 312.479,A -85,B 0,C 180,E1 -10276.676,E2 -10276.676} C_VEL
LIN {X 0,Y 424.235,Z 218.368,A -85,B 0,C 180,E1 -10278.691,E2 -10278.691} C_VEL
LIN {X 0,Y 421.118,Z 200.521,A -85,B 0,C 180,E1 -10279.242,E2 -10279.242} C_VEL
LIN {X 0,Y 422.049,Z 183.787,A -85,B 0,C 180,E1 -10282.262,E2 -10282.262} C_VEL
LIN {X 0,Y 422.811,Z 171.224,A -85,B 0,C 180,E1 -10284.554,E2 -10284.554} C_VEL
LIN {X 0,Y 420.825,Z 161.352,A -85,B 0,C 180,E1 -10286.535,E2 -10286.535} C_VEL
LIN {X 0,Y 418.287,Z 150.008,A -85,B 0,C 180,E1 -10288.885,E2 -10288.885} C_VEL
LIN {X 0,Y 418.251,Z 150.01,A -85,B 0,C 180,E1 -10292.528,E2 -10292.528} C_VEL
LIN {X 0,Y 418.264,Z 150.01,A -85,B 0,C 180,E1 -10294.841,E2 -10294.841} C_VEL
LIN {X 0,Y 418.249,Z 150.009,A -85,B 0,C 180,E1 -10298.442,E2 -10298.442} C_VEL
LIN {X 0,Y 418.239,Z 150.011,A -85,B 0,C 180,E1 -10302.234,E2 -10302.234} C_VEL
LIN {X 0,Y 418.241,Z 150.013,A -85,B 0,C 180,E1 -10305.108,E2 -10305.108} C_VEL
LIN {X 0,Y 418.245,Z 150.011,A -85,B 0,C 180,E1 -10307.766,E2 -10307.766} C_VEL
LIN {X 0,Y 418.251,Z 150.009,A -85,B 0,C 180,E1 -10310.62,E2 -10310.62} C_VEL
LIN {X 0,Y 418.247,Z 150.014,A -85,B 0,C 180,E1 -10313.975,E2 -10313.975} C_VEL
LIN {X 0,Y 418.262,Z 150.01,A -85,B 0,C 180,E1 -10317.156,E2 -10317.156} C_VEL
LIN {X 0,Y 418.259,Z 150.054,A -85,B 0,C 180,E1 -10320.18,E2 -10320.18} C_VEL
LIN {X 0,Y 422.052,Z 163.18,A -85,B 0,C 180,E1 -10322.42,E2 -10322.42} C_VEL
LIN {X 0,Y 423.107,Z 166.94,A -85,B 0,C 180,E1 -10322.976,E2 -10322.976} C_VEL
LIN {X 0,Y 429.731,Z 182.339,A -85,B 0,C 180,E1 -10323.719,E2 -10323.719} C_VEL
LIN {X 0,Y 431.19,Z 188.689,A -85,B 0,C 180,E1 -10323.933,E2 -10323.933} C_VEL
LIN {X 0,Y 429.557,Z 285.884,A -85,B 0,C 180,E1 -10325.598,E2 -10325.598} C_VEL
LIN {X 0,Y 429.101,Z 313.424,A -85,B 0,C 180,E1 -10326.069,E2 -10326.069} C_VEL
LIN {X 0,Y 428.341,Z 319.271,A -85,B 0,C 180,E1 -10326.125,E2 -10326.125} C_VEL
LIN {X 0,Y 422.72,Z 338.262,A -85,B 0,C 180,E1 -10326.19,E2 -10326.19} C_VEL
LIN {X 0,Y 421.98,Z 344.031,A -85,B 0,C 180,E1 -10326.323,E2 -10326.323} C_VEL
LIN {X 0,Y 421.373,Z 358.796,A -85,B 0,C 180,E1 -10326.886,E2 -10326.886} C_VEL
LIN {X 0,Y 420.602,Z 373.561,A -85,B 0,C 180,E1 -10327.657,E2 -10327.657} C_VEL
LIN {X 0,Y 419.522,Z 388.088,A -85,B 0,C 180,E1 -10328.63,E2 -10328.63} C_VEL
LIN {X 0,Y 418.286,Z 401.166,A -85,B 0,C 180,E1 -10329.723,E2 -10329.723} C_VEL
LIN {X 0,Y 417.022,Z 413.969,A -85,B 0,C 180,E1 -10331.035,E2 -10331.035} C_VEL
LIN {X 0,Y 415.793,Z 426.013,A -85,B 0,C 180,E1 -10332.54,E2 -10332.54} C_VEL
LIN {X 0,Y 414.642,Z 435.887,A -85,B 0,C 180,E1 -10334.011,E2 -10334.011} C_VEL
LIN {X 0,Y 413.54,Z 444.975,A -85,B 0,C 180,E1 -10335.627,E2 -10335.627} C_VEL
LIN {X 0,Y 412.605,Z 453.497,A -85,B 0,C 180,E1 -10337.456,E2 -10337.456} C_VEL
LIN {X 0,Y 411.884,Z 460.093,A -85,B 0,C 180,E1 -10339.181,E2 -10339.181} C_VEL
LIN {X 0,Y 411.251,Z 466.192,A -85,B 0,C 180,E1 -10341.151,E2 -10341.151} C_VEL
LIN {X 0,Y 410.839,Z 470.902,A -85,B 0,C 180,E1 -10343.121,E2 -10343.121} C_VEL
LIN {X 0,Y 410.643,Z 474.348,A -85,B 0,C 180,E1 -10345.09,E2 -10345.09} C_VEL
LIN {X 0,Y 410.472,Z 476.626,A -85,B 0,C 180,E1 -10347.054,E2 -10347.054} C_VEL
LIN {X 0,Y 410.188,Z 477.801,A -85,B 0,C 180,E1 -10349.017,E2 -10349.017} C_VEL
LIN {X 0,Y 410.188,Z 477.816,A -85,B 0,C 180,E1 -10350.98,E2 -10350.98} C_VEL
LIN {X 0,Y 410.47,Z 476.699,A -85,B 0,C 180,E1 -10352.943,E2 -10352.943} C_VEL
LIN {X 0,Y 410.631,Z 474.484,A -85,B 0,C 180,E1 -10354.908,E2 -10354.908} C_VEL
LIN {X 0,Y 410.837,Z 471.108,A -85,B 0,C 180,E1 -10356.876,E2 -10356.876} C_VEL
LIN {X 0,Y 411.244,Z 466.469,A -85,B 0,C 180,E1 -10358.846,E2 -10358.846} C_VEL
LIN {X 0,Y 411.87,Z 460.437,A -85,B 0,C 180,E1 -10360.817,E2 -10360.817} C_VEL
LIN {X 0,Y 412.676,Z 452.844,A -85,B 0,C 180,E1 -10362.79,E2 -10362.79} C_VEL
LIN {X 0,Y 413.61,Z 444.483,A -85,B 0,C 180,E1 -10364.562,E2 -10364.562} C_VEL
LIN {X 0,Y 414.775,Z 434.935,A -85,B 0,C 180,E1 -10366.234,E2 -10366.234} C_VEL
LIN {X 0,Y 415.913,Z 424.918,A -85,B 0,C 180,E1 -10367.706,E2 -10367.706} C_VEL
LIN {X 0,Y 417.124,Z 412.838,A -85,B 0,C 180,E1 -10369.187,E2 -10369.187} C_VEL
LIN {X 0,Y 418.34,Z 400.873,A -85,B 0,C 180,E1 -10370.4,E2 -10370.4} C_VEL
LIN {X 0,Y 419.601,Z 387.71,A -85,B 0,C 180,E1 -10371.492,E2 -10371.492} C_VEL
LIN {X 0,Y 420.571,Z 374.161,A -85,B 0,C 180,E1 -10372.407,E2 -10372.407} C_VEL
LIN {X 0,Y 421.371,Z 359.005,A -85,B 0,C 180,E1 -10373.204,E2 -10373.204} C_VEL
LIN {X 0,Y 421.992,Z 344.23,A -85,B 0,C 180,E1 -10373.769,E2 -10373.769} C_VEL
LIN {X 0,Y 422.401,Z 328.475,A -85,B 0,C 180,E1 -10374.164,E2 -10374.164} C_VEL
LIN {X 0,Y 424.87,Z 191.01,A -85,B 0,C 180,E1 -10376.549,E2 -10376.549} C_VEL
LIN {X 0,Y 424.237,Z 187.312,A -85,B 0,C 180,E1 -10376.662,E2 -10376.662} C_VEL
LIN {X 0,Y 422.861,Z 182.837,A -85,B 0,C 180,E1 -10376.842,E2 -10376.842} C_VEL
LIN {X 0,Y 415.992,Z 167.215,A -85,B 0,C 180,E1 -10377.636,E2 -10377.636} C_VEL
LIN {X 0,Y 411.971,Z 153.649,A -85,B 0,C 180,E1 -10379.903,E2 -10379.903} C_VEL
LIN {X 0,Y 411.201,Z 150.893,A -85,B 0,C 180,E1 -10380.418,E2 -10380.418} C_VEL
LIN {X 0,Y 411.202,Z 150.887,A -85,B 0,C 180,E1 -10383.154,E2 -10383.154} C_VEL
LIN {X 0,Y 411.19,Z 150.888,A -85,B 0,C 180,E1 -10386.552,E2 -10386.552} C_VEL
LIN {X 0,Y 411.205,Z 150.869,A -85,B 0,C 180,E1 -10389.726,E2 -10389.726} C_VEL
LIN {X 0,Y 411.174,Z 150.896,A -85,B 0,C 180,E1 -10393.131,E2 -10393.131} C_VEL
LIN {X 0,Y 411.161,Z 150.894,A -85,B 0,C 180,E1 -10395.88,E2 -10395.88} C_VEL
LIN {X 0,Y 411.192,Z 150.887,A -85,B 0,C 180,E1 -10398.765,E2 -10398.765} C_VEL
LIN {X 0,Y 411.197,Z 150.885,A -85,B 0,C 180,E1 -10402.026,E2 -10402.026} C_VEL
LIN {X 0,Y 411.198,Z 150.882,A -85,B 0,C 180,E1 -10405.666,E2 -10405.666} C_VEL
LIN {X 0,Y 411.193,Z 150.882,A -85,B 0,C 180,E1 -10409.153,E2 -10409.153} C_VEL
LIN {X 0,Y 411.25,Z 150.882,A -85,B 0,C 180,E1 -10412.522,E2 -10412.522} C_VEL
LIN {X 0,Y 411.21,Z 150.879,A -85,B 0,C 180,E1 -10415.783,E2 -10415.783} C_VEL
LIN {X 0,Y 411.186,Z 150.89,A -85,B 0,C 180,E1 -10418.965,E2 -10418.965} C_VEL
LIN {X 0,Y 411.242,Z 150.875,A -85,B 0,C 180,E1 -10422.084,E2 -10422.084} C_VEL
LIN {X 0,Y 411.252,Z 150.878,A -85,B 0,C 180,E1 -10425.147,E2 -10425.147} C_VEL
LIN {X 0,Y 411.275,Z 150.868,A -85,B 0,C 180,E1 -10428.167,E2 -10428.167} C_VEL
LIN {X 0,Y 411.471,Z 150.85,A -85,B 0,C 180,E1 -10432.146,E2 -10432.146} C_VEL
LIN {X 0,Y 411.464,Z 150.839,A -85,B 0,C 180,E1 -10434.118,E2 -10434.118} C_VEL
LIN {X 0,Y 411.503,Z 150.848,A -85,B 0,C 180,E1 -10438.042,E2 -10438.042} C_VEL
LIN {X 0,Y 411.632,Z 150.819,A -85,B 0,C 180,E1 -10440,E2 -10440} C_VEL
LIN {X 0,Y 411.456,Z 150.857,A -85,B 0,C 180,E1 -10442.937,E2 -10442.937} C_VEL
LIN {X 0,Y 411.449,Z 150.842,A -85,B 0,C 180,E1 -10446.867,E2 -10446.867} C_VEL
LIN {X 0,Y 411.283,Z 150.873,A -85,B 0,C 180,E1 -10449.839,E2 -10449.839} C_VEL
LIN {X 0,Y 411.294,Z 150.86,A -85,B 0,C 180,E1 -10453.104,E2 -10453.104} C_VEL
LIN {X 0,Y 411.252,Z 150.877,A -85,B 0,C 180,E1 -10455.868,E2 -10455.868} C_VEL
LIN {X 0,Y 411.214,Z 150.872,A -85,B 0,C 180,E1 -10458.949,E2 -10458.949} C_VEL
LIN {X 0,Y 411.194,Z 150.886,A -85,B 0,C 180,E1 -10462.643,E2 -10462.643} C_VEL
LIN {X 0,Y 411.226,Z 150.877,A -85,B 0,C 180,E1 -10465.294,E2 -10465.294} C_VEL
LIN {X 0,Y 411.248,Z 150.881,A -85,B 0,C 180,E1 -10467.478,E2 -10467.478} C_VEL
LIN {X 0,Y 411.179,Z 150.89,A -85,B 0,C 180,E1 -10470.848,E2 -10470.848} C_VEL
LIN {X 0,Y 411.196,Z 150.883,A -85,B 0,C 180,E1 -10474.334,E2 -10474.334} C_VEL
LIN {X 0,Y 411.191,Z 150.882,A -85,B 0,C 180,E1 -10477.974,E2 -10477.974} C_VEL
LIN {X 0,Y 411.172,Z 150.861,A -85,B 0,C 180,E1 -10480.505,E2 -10480.505} C_VEL
LIN {X 0,Y 411.164,Z 150.89,A -85,B 0,C 180,E1 -10483.135,E2 -10483.135} C_VEL
LIN {X 0,Y 411.228,Z 150.888,A -85,B 0,C 180,E1 -10485.872,E2 -10485.872} C_VEL
LIN {X 0,Y 411.203,Z 150.889,A -85,B 0,C 180,E1 -10488.765,E2 -10488.765} C_VEL
LIN {X 0,Y 411.197,Z 150.886,A -85,B 0,C 180,E1 -10492.029,E2 -10492.029} C_VEL
LIN {X 0,Y 411.22,Z 150.95,A -85,B 0,C 180,E1 -10492.891,E2 -10492.891} C_VEL
LIN {X 0,Y 418.08,Z 173.589,A -85,B 0,C 180,E1 -10496.309,E2 -10496.309} C_VEL
LIN {X 0,Y 421.658,Z 186.088,A -85,B 0,C 180,E1 -10498.094,E2 -10498.094} C_VEL
LIN {X 0,Y 419.35,Z 211.641,A -85,B 0,C 180,E1 -10501.06,E2 -10501.06} C_VEL
LIN {X 0,Y 418.089,Z 226.509,A -85,B 0,C 180,E1 -10502.764,E2 -10502.764} C_VEL
LIN {X 0,Y 423.002,Z 266.244,A -85,B 0,C 180,E1 -10503.834,E2 -10503.834} C_VEL
LIN {X 0,Y 421.57,Z 355.076,A -85,B 0,C 180,E1 -10505.37,E2 -10505.37} C_VEL
LIN {X 0,Y 420.741,Z 400.215,A -85,B 0,C 180,E1 -10506.172,E2 -10506.172} C_VEL
LIN {X 0,Y 419.933,Z 416.232,A -85,B 0,C 180,E1 -10506.646,E2 -10506.646} C_VEL
LIN {X 0,Y 418.844,Z 431.382,A -85,B 0,C 180,E1 -10507.3,E2 -10507.3} C_VEL
LIN {X 0,Y 417.671,Z 446.421,A -85,B 0,C 180,E1 -10508.178,E2 -10508.178} C_VEL
LIN {X 0,Y 416.231,Z 460.705,A -85,B 0,C 180,E1 -10509.234,E2 -10509.234} C_VEL
LIN {X 0,Y 414.996,Z 474.008,A -85,B 0,C 180,E1 -10510.461,E2 -10510.461} C_VEL
LIN {X 0,Y 413.776,Z 485.539,A -85,B 0,C 180,E1 -10511.739,E2 -10511.739} C_VEL
LIN {X 0,Y 412.781,Z 496.409,A -85,B 0,C 180,E1 -10513.177,E2 -10513.177} C_VEL
LIN {X 0,Y 411.728,Z 507.34,A -85,B 0,C 180,E1 -10514.913,E2 -10514.913} C_VEL
LIN {X 0,Y 411.055,Z 516.45,A -85,B 0,C 180,E1 -10516.656,E2 -10516.656} C_VEL
LIN {X 0,Y 410.623,Z 522.999,A -85,B 0,C 180,E1 -10518.149,E2 -10518.149} C_VEL
LIN {X 0,Y 410.269,Z 530.259,A -85,B 0,C 180,E1 -10520.138,E2 -10520.138} C_VEL
LIN {X 0,Y 410.207,Z 535.983,A -85,B 0,C 180,E1 -10522.123,E2 -10522.123} C_VEL
LIN {X 0,Y 410.272,Z 540.311,A -85,B 0,C 180,E1 -10524.102,E2 -10524.102} C_VEL
LIN {X 0,Y 410.339,Z 543.346,A -85,B 0,C 180,E1 -10526.073,E2 -10526.073} C_VEL
LIN {X 0,Y 410.356,Z 545.155,A -85,B 0,C 180,E1 -10528.038,E2 -10528.038} C_VEL
LIN {X 0,Y 410.351,Z 545.771,A -85,B 0,C 180,E1 -10530.001,E2 -10530.001} C_VEL
LIN {X 0,Y 410.357,Z 545.154,A -85,B 0,C 180,E1 -10531.964,E2 -10531.964} C_VEL
LIN {X 0,Y 410.337,Z 543.343,A -85,B 0,C 180,E1 -10533.93,E2 -10533.93} C_VEL
LIN {X 0,Y 410.276,Z 540.3,A -85,B 0,C 180,E1 -10535.9,E2 -10535.9} C_VEL
LIN {X 0,Y 410.246,Z 535.964,A -85,B 0,C 180,E1 -10537.878,E2 -10537.878} C_VEL
LIN {X 0,Y 410.321,Z 530.238,A -85,B 0,C 180,E1 -10539.863,E2 -10539.863} C_VEL
LIN {X 0,Y 410.667,Z 522.977,A -85,B 0,C 180,E1 -10541.852,E2 -10541.852} C_VEL
LIN {X 0,Y 411.139,Z 515.327,A -85,B 0,C 180,E1 -10543.57,E2 -10543.57} C_VEL
LIN {X 0,Y 411.873,Z 505.849,A -85,B 0,C 180,E1 -10545.337,E2 -10545.337} C_VEL
LIN {X 0,Y 412.805,Z 496.355,A -85,B 0,C 180,E1 -10546.825,E2 -10546.825} C_VEL
LIN {X 0,Y 413.801,Z 485.074,A -85,B 0,C 180,E1 -10548.313,E2 -10548.313} C_VEL
LIN {X 0,Y 415.043,Z 472.724,A -85,B 0,C 180,E1 -10549.668,E2 -10549.668} C_VEL
LIN {X 0,Y 416.414,Z 459.163,A -85,B 0,C 180,E1 -10550.889,E2 -10550.889} C_VEL
LIN {X 0,Y 417.804,Z 444.817,A -85,B 0,C 180,E1 -10551.923,E2 -10551.923} C_VEL
LIN {X 0,Y 418.902,Z 431.204,A -85,B 0,C 180,E1 -10552.699,E2 -10552.699} C_VEL
LIN {X 0,Y 419.968,Z 415.973,A -85,B 0,C 180,E1 -10553.354,E2 -10553.354} C_VEL
LIN {X 0,Y 420.739,Z 401.055,A -85,B 0,C 180,E1 -10553.799,E2 -10553.799} C_VEL
LIN {X 0,Y 421.542,Z 361.693,A -85,B 0,C 180,E1 -10554.503,E2 -10554.503} C_VEL
LIN {X 0,Y 422.605,Z 298.254,A -85,B 0,C 180,E1 -10555.62,E2 -10555.62} C_VEL
LIN {X 0,Y 423.804,Z 265.895,A -85,B 0,C 180,E1 -10556.386,E2 -10556.386} C_VEL
LIN {X 0,Y 421.773,Z 244.282,A -85,B 0,C 180,E1 -10557.171,E2 -10557.171} C_VEL
LIN {X 0,Y 420.334,Z 234.321,A -85,B 0,C 180,E1 -10557.605,E2 -10557.605} C_VEL
LIN {X 0,Y 424,Z 208.772,A -85,B 0,C 180,E1 -10560.921,E2 -10560.921} C_VEL
LIN {X 0,Y 426.706,Z 194.223,A -85,B 0,C 180,E1 -10562.925,E2 -10562.925} C_VEL
LIN {X 0,Y 425.078,Z 186.927,A -85,B 0,C 180,E1 -10564.423,E2 -10564.423} C_VEL
LIN {X 0,Y 422.786,Z 179.4,A -85,B 0,C 180,E1 -10566.273,E2 -10566.273} C_VEL
LIN {X 0,Y 420.482,Z 172.892,A -85,B 0,C 180,E1 -10568.227,E2 -10568.227} C_VEL
LIN {X 0,Y 418.475,Z 167.782,A -85,B 0,C 180,E1 -10570.153,E2 -10570.153} C_VEL
LIN {X 0,Y 416.8,Z 163.879,A -85,B 0,C 180,E1 -10572.105,E2 -10572.105} C_VEL
LIN {X 0,Y 415.7,Z 161.382,A -85,B 0,C 180,E1 -10573.882,E2 -10573.882} C_VEL
LIN {X 0,Y 414.934,Z 159.553,A -85,B 0,C 180,E1 -10576.017,E2 -10576.017} C_VEL
LIN {X 0,Y 414.807,Z 158.995,A -85,B 0,C 180,E1 -10577.335,E2 -10577.335} C_VEL
LIN {X 0,Y 414.72,Z 159.048,A -85,B 0,C 180,E1 -10578.631,E2 -10578.631} C_VEL
LIN {X 0,Y 415.094,Z 160.518,A -85,B 0,C 180,E1 -10581.211,E2 -10581.211} C_VEL
LIN {X 0,Y 415.684,Z 161.926,A -85,B 0,C 180,E1 -10582.622,E2 -10582.622} C_VEL
LIN {X 0,Y 417.041,Z 165.486,A -85,B 0,C 180,E1 -10585.043,E2 -10585.043} C_VEL
LIN {X 0,Y 418.395,Z 169.665,A -85,B 0,C 180,E1 -10587.128,E2 -10587.128} C_VEL
LIN {X 0,Y 420.08,Z 175.657,A -85,B 0,C 180,E1 -10589.517,E2 -10589.517} C_VEL
LIN {X 0,Y 421.978,Z 183.774,A -85,B 0,C 180,E1 -10592.203,E2 -10592.203} C_VEL
LIN {X 0,Y 422.886,Z 189.469,A -85,B 0,C 180,E1 -10593.824,E2 -10593.824} C_VEL
LIN {X 0,Y 422.626,Z 192.928,A -85,B 0,C 180,E1 -10594.646,E2 -10594.646} C_VEL
LIN {X 0,Y 420.236,Z 208.318,A -85,B 0,C 180,E1 -10597.928,E2 -10597.928} C_VEL
LIN {X 0,Y 424.351,Z 224.196,A -85,B 0,C 180,E1 -10598.933,E2 -10598.933} C_VEL
LIN {X 0,Y 424.704,Z 226.791,A -85,B 0,C 180,E1 -10599.058,E2 -10599.058} C_VEL
LIN {X 0,Y 419.779,Z 313.78,A -85,B 0,C 180,E1 -10601.578,E2 -10601.578} C_VEL
LIN {X 0,Y 419.3,Z 329.768,A -85,B 0,C 180,E1 -10602.094,E2 -10602.094} C_VEL
LIN {X 0,Y 418.779,Z 342.901,A -85,B 0,C 180,E1 -10602.695,E2 -10602.695} C_VEL
LIN {X 0,Y 418.006,Z 357.247,A -85,B 0,C 180,E1 -10603.582,E2 -10603.582} C_VEL
LIN {X 0,Y 417.247,Z 368.695,A -85,B 0,C 180,E1 -10604.491,E2 -10604.491} C_VEL
LIN {X 0,Y 416.351,Z 380.877,A -85,B 0,C 180,E1 -10605.708,E2 -10605.708} C_VEL
LIN {X 0,Y 415.62,Z 389.822,A -85,B 0,C 180,E1 -10606.804,E2 -10606.804} C_VEL
LIN {X 0,Y 414.882,Z 398.116,A -85,B 0,C 180,E1 -10608.024,E2 -10608.024} C_VEL
LIN {X 0,Y 414.054,Z 406.247,A -85,B 0,C 180,E1 -10609.487,E2 -10609.487} C_VEL
LIN {X 0,Y 413.165,Z 413.757,A -85,B 0,C 180,E1 -10611.194,E2 -10611.194} C_VEL
LIN {X 0,Y 412.71,Z 418.735,A -85,B 0,C 180,E1 -10612.662,E2 -10612.662} C_VEL
LIN {X 0,Y 412.165,Z 422.572,A -85,B 0,C 180,E1 -10614.128,E2 -10614.128} C_VEL
LIN {X 0,Y 411.958,Z 424.52,A -85,B 0,C 180,E1 -10615.107,E2 -10615.107} C_VEL
LIN {X 0,Y 411.798,Z 425.995,A -85,B 0,C 180,E1 -10616.086,E2 -10616.086} C_VEL
LIN {X 0,Y 411.606,Z 427.064,A -85,B 0,C 180,E1 -10617.064,E2 -10617.064} C_VEL
LIN {X 0,Y 411.509,Z 427.713,A -85,B 0,C 180,E1 -10618.043,E2 -10618.043} C_VEL
LIN {X 0,Y 411.331,Z 427.933,A -85,B 0,C 180,E1 -10619.021,E2 -10619.021} C_VEL
LIN {X 0,Y 411.253,Z 427.707,A -85,B 0,C 180,E1 -10620,E2 -10620} C_VEL
LIN {X 0,Y 411.268,Z 427.07,A -85,B 0,C 180,E1 -10620.979,E2 -10620.979} C_VEL
LIN {X 0,Y 411.188,Z 426.048,A -85,B 0,C 180,E1 -10621.959,E2 -10621.959} C_VEL
LIN {X 0,Y 411.302,Z 424.545,A -85,B 0,C 180,E1 -10622.938,E2 -10622.938} C_VEL
LIN {X 0,Y 411.268,Z 421.512,A -85,B 0,C 180,E1 -10624.41,E2 -10624.41} C_VEL
LIN {X 0,Y 411.527,Z 417.395,A -85,B 0,C 180,E1 -10625.881,E2 -10625.881} C_VEL
LIN {X 0,Y 411.839,Z 411.121,A -85,B 0,C 180,E1 -10627.6,E2 -10627.6} C_VEL
LIN {X 0,Y 412.115,Z 404.323,A -85,B 0,C 180,E1 -10629.076,E2 -10629.076} C_VEL
LIN {X 0,Y 412.556,Z 395.911,A -85,B 0,C 180,E1 -10630.552,E2 -10630.552} C_VEL
LIN {X 0,Y 413.072,Z 385.454,A -85,B 0,C 180,E1 -10632.03,E2 -10632.03} C_VEL
LIN {X 0,Y 413.593,Z 374.695,A -85,B 0,C 180,E1 -10633.262,E2 -10633.262} C_VEL
LIN {X 0,Y 414.222,Z 361.973,A -85,B 0,C 180,E1 -10634.426,E2 -10634.426} C_VEL
LIN {X 0,Y 414.645,Z 349.684,A -85,B 0,C 180,E1 -10635.32,E2 -10635.32} C_VEL
LIN {X 0,Y 415.063,Z 335.62,A -85,B 0,C 180,E1 -10636.097,E2 -10636.097} C_VEL
LIN {X 0,Y 415.407,Z 322.619,A -85,B 0,C 180,E1 -10636.62,E2 -10636.62} C_VEL
LIN {X 0,Y 415.627,Z 305.687,A -85,B 0,C 180,E1 -10637.054,E2 -10637.054} C_VEL
LIN {X 0,Y 417.447,Z 219.497,A -85,B 0,C 180,E1 -10638.945,E2 -10638.945} C_VEL
LIN {X 0,Y 414.253,Z 200.768,A -85,B 0,C 180,E1 -10639.536,E2 -10639.536} C_VEL
LIN {X 0,Y 415.368,Z 182.319,A -85,B 0,C 180,E1 -10642.902,E2 -10642.902} C_VEL
LIN {X 0,Y 415.919,Z 172.615,A -85,B 0,C 180,E1 -10644.699,E2 -10644.699} C_VEL
LIN {X 0,Y 413.592,Z 161.161,A -85,B 0,C 180,E1 -10647.036,E2 -10647.036} C_VEL
LIN {X 0,Y 411.235,Z 150.888,A -85,B 0,C 180,E1 -10649.209,E2 -10649.209} C_VEL
LIN {X 0,Y 411.171,Z 150.893,A -85,B 0,C 180,E1 -10651.997,E2 -10651.997} C_VEL
LIN {X 0,Y 411.216,Z 150.888,A -85,B 0,C 180,E1 -10654.878,E2 -10654.878} C_VEL
LIN {X 0,Y 411.203,Z 150.887,A -85,B 0,C 180,E1 -10658.167,E2 -10658.167} C_VEL
LIN {X 0,Y 411.163,Z 150.893,A -85,B 0,C 180,E1 -10661.227,E2 -10661.227} C_VEL
LIN {X 0,Y 411.18,Z 150.886,A -85,B 0,C 180,E1 -10664.49,E2 -10664.49} C_VEL
LIN {X 0,Y 411.182,Z 150.89,A -85,B 0,C 180,E1 -10668.194,E2 -10668.194} C_VEL
LIN {X 0,Y 411.216,Z 150.887,A -85,B 0,C 180,E1 -10670.775,E2 -10670.775} C_VEL
LIN {X 0,Y 411.202,Z 150.892,A -85,B 0,C 180,E1 -10674.47,E2 -10674.47} C_VEL
LIN {X 0,Y 411.212,Z 150.888,A -85,B 0,C 180,E1 -10676.873,E2 -10676.873} C_VEL
LIN {X 0,Y 411.22,Z 151.008,A -85,B 0,C 180,E1 -10679.722,E2 -10679.722} C_VEL
LIN {X 0,Y 415.377,Z 165.061,A -85,B 0,C 180,E1 -10682.132,E2 -10682.132} C_VEL
LIN {X 0,Y 416.087,Z 167.505,A -85,B 0,C 180,E1 -10682.483,E2 -10682.483} C_VEL
LIN {X 0,Y 423.563,Z 184.528,A -85,B 0,C 180,E1 -10683.338,E2 -10683.338} C_VEL
LIN {X 0,Y 424.883,Z 190.392,A -85,B 0,C 180,E1 -10683.539,E2 -10683.539} C_VEL
LIN {X 0,Y 422.257,Z 333.58,A -85,B 0,C 180,E1 -10686.042,E2 -10686.042} C_VEL
LIN {X 0,Y 421.98,Z 344.031,A -85,B 0,C 180,E1 -10686.323,E2 -10686.323} C_VEL
LIN {X 0,Y 421.153,Z 349.785,A -85,B 0,C 180,E1 -10686.474,E2 -10686.474} C_VEL
LIN {X 0,Y 418.093,Z 359.094,A -85,B 0,C 180,E1 -10686.693,E2 -10686.693} C_VEL
LIN {X 0,Y 414.994,Z 368.32,A -85,B 0,C 180,E1 -10686.987,E2 -10686.987} C_VEL
LIN {X 0,Y 414.075,Z 373.718,A -85,B 0,C 180,E1 -10687.26,E2 -10687.26} C_VEL
LIN {X 0,Y 413.076,Z 386.966,A -85,B 0,C 180,E1 -10688.149,E2 -10688.149} C_VEL
LIN {X 0,Y 411.813,Z 400.365,A -85,B 0,C 180,E1 -10689.259,E2 -10689.259} C_VEL
LIN {X 0,Y 410.49,Z 412.555,A -85,B 0,C 180,E1 -10690.491,E2 -10690.491} C_VEL
LIN {X 0,Y 409.481,Z 422.863,A -85,B 0,C 180,E1 -10691.745,E2 -10691.745} C_VEL
LIN {X 0,Y 408.223,Z 433.321,A -85,B 0,C 180,E1 -10693.238,E2 -10693.238} C_VEL
LIN {X 0,Y 406.917,Z 443.492,A -85,B 0,C 180,E1 -10694.984,E2 -10694.984} C_VEL
LIN {X 0,Y 405.959,Z 451.924,A -85,B 0,C 180,E1 -10696.738,E2 -10696.738} C_VEL
LIN {X 0,Y 405.125,Z 458.934,A -85,B 0,C 180,E1 -10698.491,E2 -10698.491} C_VEL
LIN {X 0,Y 404.434,Z 465.404,A -85,B 0,C 180,E1 -10700.497,E2 -10700.497} C_VEL
LIN {X 0,Y 403.893,Z 470.816,A -85,B 0,C 180,E1 -10702.675,E2 -10702.675} C_VEL
LIN {X 0,Y 403.587,Z 473.37,A -85,B 0,C 180,E1 -10704.001,E2 -10704.001} C_VEL
LIN {X 0,Y 403.484,Z 476.215,A -85,B 0,C 180,E1 -10706.004,E2 -10706.004} C_VEL
LIN {X 0,Y 403.243,Z 477.936,A -85,B 0,C 180,E1 -10708.001,E2 -10708.001} C_VEL
LIN {X 0,Y 403.104,Z 478.538,A -85,B 0,C 180,E1 -10709.999,E2 -10709.999} C_VEL
LIN {X 0,Y 403.242,Z 477.98,A -85,B 0,C 180,E1 -10711.996,E2 -10711.996} C_VEL
LIN {X 0,Y 403.479,Z 476.317,A -85,B 0,C 180,E1 -10713.994,E2 -10713.994} C_VEL
LIN {X 0,Y 403.567,Z 473.54,A -85,B 0,C 180,E1 -10715.996,E2 -10715.996} C_VEL
LIN {X 0,Y 404.026,Z 469.535,A -85,B 0,C 180,E1 -10717.998,E2 -10717.998} C_VEL
LIN {X 0,Y 404.573,Z 464.217,A -85,B 0,C 180,E1 -10720.002,E2 -10720.002} C_VEL
LIN {X 0,Y 405.307,Z 457.431,A -85,B 0,C 180,E1 -10722.008,E2 -10722.008} C_VEL
LIN {X 0,Y 406.203,Z 450.149,A -85,B 0,C 180,E1 -10723.761,E2 -10723.761} C_VEL
LIN {X 0,Y 407.233,Z 441.365,A -85,B 0,C 180,E1 -10725.514,E2 -10725.514} C_VEL
LIN {X 0,Y 408.501,Z 430.723,A -85,B 0,C 180,E1 -10727.263,E2 -10727.263} C_VEL
LIN {X 0,Y 409.777,Z 419.776,A -85,B 0,C 180,E1 -10728.757,E2 -10728.757} C_VEL
LIN {X 0,Y 411.094,Z 407.741,A -85,B 0,C 180,E1 -10730.123,E2 -10730.123} C_VEL
LIN {X 0,Y 412.446,Z 394.436,A -85,B 0,C 180,E1 -10731.358,E2 -10731.358} C_VEL
LIN {X 0,Y 413.56,Z 381.413,A -85,B 0,C 180,E1 -10732.347,E2 -10732.347} C_VEL
LIN {X 0,Y 414.507,Z 368.264,A -85,B 0,C 180,E1 -10733.148,E2 -10733.148} C_VEL
LIN {X 0,Y 415.177,Z 354.005,A -85,B 0,C 180,E1 -10733.825,E2 -10733.825} C_VEL
LIN {X 0,Y 415.71,Z 338.945,A -85,B 0,C 180,E1 -10734.334,E2 -10734.334} C_VEL
LIN {X 0,Y 416.123,Z 318.997,A -85,B 0,C 180,E1 -10734.74,E2 -10734.74} C_VEL
LIN {X 0,Y 418.557,Z 191.885,A -85,B 0,C 180,E1 -10736.974,E2 -10736.974} C_VEL
LIN {X 0,Y 417.103,Z 186.141,A -85,B 0,C 180,E1 -10737.187,E2 -10737.187} C_VEL
LIN {X 0,Y 408.933,Z 167.673,A -85,B 0,C 180,E1 -10738.167,E2 -10738.167} C_VEL
LIN {X 0,Y 404.734,Z 153.773,A -85,B 0,C 180,E1 -10740.523,E2 -10740.523} C_VEL
LIN {X 0,Y 404.138,Z 151.77,A -85,B 0,C 180,E1 -10740.935,E2 -10740.935} C_VEL
LIN {X 0,Y 404.14,Z 151.772,A -85,B 0,C 180,E1 -10743.811,E2 -10743.811} C_VEL
LIN {X 0,Y 404.134,Z 151.767,A -85,B 0,C 180,E1 -10746.874,E2 -10746.874} C_VEL
LIN {X 0,Y 404.141,Z 151.746,A -85,B 0,C 180,E1 -10750.079,E2 -10750.079} C_VEL
LIN {X 0,Y 404.154,Z 151.77,A -85,B 0,C 180,E1 -10753.084,E2 -10753.084} C_VEL
LIN {X 0,Y 404.141,Z 151.768,A -85,B 0,C 180,E1 -10755.925,E2 -10755.925} C_VEL
LIN {X 0,Y 404.144,Z 151.765,A -85,B 0,C 180,E1 -10758.638,E2 -10758.638} C_VEL
LIN {X 0,Y 404.154,Z 151.761,A -85,B 0,C 180,E1 -10761.489,E2 -10761.489} C_VEL
LIN {X 0,Y 404.177,Z 151.757,A -85,B 0,C 180,E1 -10764.983,E2 -10764.983} C_VEL
LIN {X 0,Y 404.142,Z 151.767,A -85,B 0,C 180,E1 -10768.554,E2 -10768.554} C_VEL
LIN {X 0,Y 404.189,Z 151.76,A -85,B 0,C 180,E1 -10772,E2 -10772} C_VEL
LIN {X 0,Y 404.164,Z 151.754,A -85,B 0,C 180,E1 -10775.333,E2 -10775.333} C_VEL
LIN {X 0,Y 404.128,Z 151.77,A -85,B 0,C 180,E1 -10778.58,E2 -10778.58} C_VEL
LIN {X 0,Y 404.199,Z 151.752,A -85,B 0,C 180,E1 -10781.761,E2 -10781.761} C_VEL
LIN {X 0,Y 404.198,Z 151.76,A -85,B 0,C 180,E1 -10784.882,E2 -10784.882} C_VEL
LIN {X 0,Y 404.247,Z 151.743,A -85,B 0,C 180,E1 -10787.958,E2 -10787.958} C_VEL
LIN {X 0,Y 404.422,Z 151.728,A -85,B 0,C 180,E1 -10792.099,E2 -10792.099} C_VEL
LIN {X 0,Y 404.413,Z 151.717,A -85,B 0,C 180,E1 -10794.015,E2 -10794.015} C_VEL
LIN {X 0,Y 404.472,Z 151.724,A -85,B 0,C 180,E1 -10798.008,E2 -10798.008} C_VEL
LIN {X 0,Y 404.602,Z 151.694,A -85,B 0,C 180,E1 -10800,E2 -10800} C_VEL
LIN {X 0,Y 404.413,Z 151.734,A -85,B 0,C 180,E1 -10802.988,E2 -10802.988} C_VEL
LIN {X 0,Y 404.4,Z 151.719,A -85,B 0,C 180,E1 -10806.987,E2 -10806.987} C_VEL
LIN {X 0,Y 404.248,Z 151.751,A -85,B 0,C 180,E1 -10810.012,E2 -10810.012} C_VEL
LIN {X 0,Y 404.255,Z 151.736,A -85,B 0,C 180,E1 -10813.212,E2 -10813.212} C_VEL
LIN {X 0,Y 404.208,Z 151.753,A -85,B 0,C 180,E1 -10817.009,E2 -10817.009} C_VEL
LIN {X 0,Y 404.153,Z 151.758,A -85,B 0,C 180,E1 -10820.352,E2 -10820.352} C_VEL
LIN {X 0,Y 404.159,Z 151.758,A -85,B 0,C 180,E1 -10823.575,E2 -10823.575} C_VEL
LIN {X 0,Y 404.173,Z 151.756,A -85,B 0,C 180,E1 -10825.767,E2 -10825.767} C_VEL
LIN {X 0,Y 404.185,Z 151.764,A -85,B 0,C 180,E1 -10828,E2 -10828} C_VEL
LIN {X 0,Y 404.129,Z 151.767,A -85,B 0,C 180,E1 -10831.559,E2 -10831.559} C_VEL
LIN {X 0,Y 404.176,Z 151.759,A -85,B 0,C 180,E1 -10835.017,E2 -10835.017} C_VEL
LIN {X 0,Y 404.148,Z 151.749,A -85,B 0,C 180,E1 -10838.757,E2 -10838.757} C_VEL
LIN {X 0,Y 404.114,Z 151.75,A -85,B 0,C 180,E1 -10841.601,E2 -10841.601} C_VEL
LIN {X 0,Y 404.145,Z 151.769,A -85,B 0,C 180,E1 -10844.524,E2 -10844.524} C_VEL
LIN {X 0,Y 404.203,Z 151.76,A -85,B 0,C 180,E1 -10847.307,E2 -10847.307} C_VEL
LIN {X 0,Y 404.161,Z 151.766,A -85,B 0,C 180,E1 -10849.957,E2 -10849.957} C_VEL
LIN {X 0,Y 404.18,Z 151.845,A -85,B 0,C 180,E1 -10852.456,E2 -10852.456} C_VEL
LIN {X 0,Y 411.118,Z 174.87,A -85,B 0,C 180,E1 -10856.005,E2 -10856.005} C_VEL
LIN {X 0,Y 414.853,Z 187.83,A -85,B 0,C 180,E1 -10857.892,E2 -10857.892} C_VEL
LIN {X 0,Y 413.043,Z 207.321,A -85,B 0,C 180,E1 -10860.201,E2 -10860.201} C_VEL
LIN {X 0,Y 411.422,Z 224.924,A -85,B 0,C 180,E1 -10862.261,E2 -10862.261} C_VEL
LIN {X 0,Y 416.62,Z 267.191,A -85,B 0,C 180,E1 -10863.428,E2 -10863.428} C_VEL
LIN {X 0,Y 415.133,Z 354.629,A -85,B 0,C 180,E1 -10864.962,E2 -10864.962} C_VEL
LIN {X 0,Y 414.266,Z 399.727,A -85,B 0,C 180,E1 -10865.775,E2 -10865.775} C_VEL
LIN {X 0,Y 413.384,Z 415.694,A -85,B 0,C 180,E1 -10866.254,E2 -10866.254} C_VEL
LIN {X 0,Y 412.283,Z 430.829,A -85,B 0,C 180,E1 -10866.918,E2 -10866.918} C_VEL
LIN {X 0,Y 411.168,Z 444.841,A -85,B 0,C 180,E1 -10867.739,E2 -10867.739} C_VEL
LIN {X 0,Y 409.711,Z 458.697,A -85,B 0,C 180,E1 -10868.756,E2 -10868.756} C_VEL
LIN {X 0,Y 408.314,Z 472.242,A -85,B 0,C 180,E1 -10869.997,E2 -10869.997} C_VEL
LIN {X 0,Y 406.994,Z 484.561,A -85,B 0,C 180,E1 -10871.371,E2 -10871.371} C_VEL
LIN {X 0,Y 405.88,Z 495.821,A -85,B 0,C 180,E1 -10872.882,E2 -10872.882} C_VEL
LIN {X 0,Y 404.9,Z 505.309,A -85,B 0,C 180,E1 -10874.394,E2 -10874.394} C_VEL
LIN {X 0,Y 404.148,Z 514.647,A -85,B 0,C 180,E1 -10876.168,E2 -10876.168} C_VEL
LIN {X 0,Y 403.572,Z 522.407,A -85,B 0,C 180,E1 -10877.939,E2 -10877.939} C_VEL
LIN {X 0,Y 403.201,Z 529.668,A -85,B 0,C 180,E1 -10879.963,E2 -10879.963} C_VEL
LIN {X 0,Y 403.131,Z 535.394,A -85,B 0,C 180,E1 -10881.984,E2 -10881.984} C_VEL
LIN {X 0,Y 403.176,Z 539.722,A -85,B 0,C 180,E1 -10883.998,E2 -10883.998} C_VEL
LIN {X 0,Y 403.244,Z 542.758,A -85,B 0,C 180,E1 -10886.004,E2 -10886.004} C_VEL
LIN {X 0,Y 403.3,Z 544.572,A -85,B 0,C 180,E1 -10888.004,E2 -10888.004} C_VEL
LIN {X 0,Y 403.283,Z 545.187,A -85,B 0,C 180,E1 -10890.001,E2 -10890.001} C_VEL
LIN {X 0,Y 403.301,Z 544.571,A -85,B 0,C 180,E1 -10891.999,E2 -10891.999} C_VEL
LIN {X 0,Y 403.241,Z 542.755,A -85,B 0,C 180,E1 -10893.999,E2 -10893.999} C_VEL
LIN {X 0,Y 403.186,Z 539.711,A -85,B 0,C 180,E1 -10896.005,E2 -10896.005} C_VEL
LIN {X 0,Y 403.165,Z 535.374,A -85,B 0,C 180,E1 -10898.018,E2 -10898.018} C_VEL
LIN {X 0,Y 403.245,Z 529.645,A -85,B 0,C 180,E1 -10900.038,E2 -10900.038} C_VEL
LIN {X 0,Y 403.635,Z 522.384,A -85,B 0,C 180,E1 -10902.062,E2 -10902.062} C_VEL
LIN {X 0,Y 404.151,Z 514.608,A -85,B 0,C 180,E1 -10903.835,E2 -10903.835} C_VEL
LIN {X 0,Y 404.935,Z 505.257,A -85,B 0,C 180,E1 -10905.607,E2 -10905.607} C_VEL
LIN {X 0,Y 405.895,Z 495.762,A -85,B 0,C 180,E1 -10907.12,E2 -10907.12} C_VEL
LIN {X 0,Y 406.97,Z 484.48,A -85,B 0,C 180,E1 -10908.633,E2 -10908.633} C_VEL
LIN {X 0,Y 408.317,Z 472.141,A -85,B 0,C 180,E1 -10910.005,E2 -10910.005} C_VEL
LIN {X 0,Y 409.718,Z 458.582,A -85,B 0,C 180,E1 -10911.246,E2 -10911.246} C_VEL
LIN {X 0,Y 411.135,Z 444.518,A -85,B 0,C 180,E1 -10912.278,E2 -10912.278} C_VEL
LIN {X 0,Y 412.424,Z 429.421,A -85,B 0,C 180,E1 -10913.142,E2 -10913.142} C_VEL
LIN {X 0,Y 413.46,Z 414.567,A -85,B 0,C 180,E1 -10913.778,E2 -10913.778} C_VEL
LIN {X 0,Y 414.295,Z 399.241,A -85,B 0,C 180,E1 -10914.225,E2 -10914.225} C_VEL
LIN {X 0,Y 416.053,Z 310.661,A -85,B 0,C 180,E1 -10915.818,E2 -10915.818} C_VEL
LIN {X 0,Y 417.817,Z 266.847,A -85,B 0,C 180,E1 -10916.885,E2 -10916.885} C_VEL
LIN {X 0,Y 415.913,Z 245.669,A -85,B 0,C 180,E1 -10917.688,E2 -10917.688} C_VEL
LIN {X 0,Y 414.223,Z 233.764,A -85,B 0,C 180,E1 -10918.243,E2 -10918.243} C_VEL
LIN {X 0,Y 417.975,Z 210.016,A -85,B 0,C 180,E1 -10921.417,E2 -10921.417} C_VEL
LIN {X 0,Y 420.567,Z 196.613,A -85,B 0,C 180,E1 -10923.328,E2 -10923.328} C_VEL
LIN {X 0,Y 418.474,Z 187.976,A -85,B 0,C 180,E1 -10925.252,E2 -10925.252} C_VEL
LIN {X 0,Y 416.411,Z 181.41,A -85,B 0,C 180,E1 -10927.023,E2 -10927.023} C_VEL
LIN {X 0,Y 414.43,Z 175.773,A -85,B 0,C 180,E1 -10928.864,E2 -10928.864} C_VEL
LIN {X 0,Y 412.571,Z 170.974,A -85,B 0,C 180,E1 -10930.855,E2 -10930.855} C_VEL
LIN {X 0,Y 410.868,Z 167.039,A -85,B 0,C 180,E1 -10933.175,E2 -10933.175} C_VEL
LIN {X 0,Y 409.848,Z 164.801,A -85,B 0,C 180,E1 -10935.327,E2 -10935.327} C_VEL
LIN {X 0,Y 409.63,Z 163.956,A -85,B 0,C 180,E1 -10936.664,E2 -10936.664} C_VEL
LIN {X 0,Y 409.494,Z 163.701,A -85,B 0,C 180,E1 -10937.984,E2 -10937.984} C_VEL
LIN {X 0,Y 409.43,Z 163.996,A -85,B 0,C 180,E1 -10939.286,E2 -10939.286} C_VEL
LIN {X 0,Y 409.977,Z 165.914,A -85,B 0,C 180,E1 -10942.052,E2 -10942.052} C_VEL
LIN {X 0,Y 411.123,Z 168.988,A -85,B 0,C 180,E1 -10944.464,E2 -10944.464} C_VEL
LIN {X 0,Y 412.608,Z 173.645,A -85,B 0,C 180,E1 -10946.971,E2 -10946.971} C_VEL
LIN {X 0,Y 414.18,Z 179.47,A -85,B 0,C 180,E1 -10949.399,E2 -10949.399} C_VEL
LIN {X 0,Y 415.858,Z 187.029,A -85,B 0,C 180,E1 -10951.981,E2 -10951.981} C_VEL
LIN {X 0,Y 416.7,Z 193.219,A -85,B 0,C 180,E1 -10953.788,E2 -10953.788} C_VEL
LIN {X 0,Y 415.28,Z 201.997,A -85,B 0,C 180,E1 -10955.77,E2 -10955.77} C_VEL
LIN {X 0,Y 414.174,Z 209.153,A -85,B 0,C 180,E1 -10957.292,E2 -10957.292} C_VEL
LIN {X 0,Y 418.136,Z 224.264,A -85,B 0,C 180,E1 -10958.312,E2 -10958.312} C_VEL
LIN {X 0,Y 418.867,Z 228.357,A -85,B 0,C 180,E1 -10958.543,E2 -10958.543} C_VEL
LIN {X 0,Y 413.495,Z 315.807,A -85,B 0,C 180,E1 -10961.16,E2 -10961.16} C_VEL
LIN {X 0,Y 413.002,Z 331.268,A -85,B 0,C 180,E1 -10961.683,E2 -10961.683} C_VEL
LIN {X 0,Y 412.393,Z 344.79,A -85,B 0,C 180,E1 -10962.329,E2 -10962.329} C_VEL
LIN {X 0,Y 411.556,Z 358.773,A -85,B 0,C 180,E1 -10963.221,E2 -10963.221} C_VEL
LIN {X 0,Y 410.651,Z 371.058,A -85,B 0,C 180,E1 -10964.235,E2 -10964.235} C_VEL
LIN {X 0,Y 409.729,Z 382.986,A -85,B 0,C 180,E1 -10965.472,E2 -10965.472} C_VEL
LIN {X 0,Y 408.963,Z 391.736,A -85,B 0,C 180,E1 -10966.585,E2 -10966.585} C_VEL
LIN {X 0,Y 407.999,Z 401.303,A -85,B 0,C 180,E1 -10968.071,E2 -10968.071} C_VEL
LIN {X 0,Y 407.12,Z 409.264,A -85,B 0,C 180,E1 -10969.607,E2 -10969.607} C_VEL
LIN {X 0,Y 406.312,Z 415.272,A -85,B 0,C 180,E1 -10971.044,E2 -10971.044} C_VEL
LIN {X 0,Y 405.823,Z 420.151,A -85,B 0,C 180,E1 -10972.537,E2 -10972.537} C_VEL
LIN {X 0,Y 405.243,Z 423.907,A -85,B 0,C 180,E1 -10974.027,E2 -10974.027} C_VEL
LIN {X 0,Y 405.009,Z 425.789,A -85,B 0,C 180,E1 -10975.023,E2 -10975.023} C_VEL
LIN {X 0,Y 404.821,Z 427.223,A -85,B 0,C 180,E1 -10976.018,E2 -10976.018} C_VEL
LIN {X 0,Y 404.638,Z 428.246,A -85,B 0,C 180,E1 -10977.013,E2 -10977.013} C_VEL
LIN {X 0,Y 404.518,Z 428.847,A -85,B 0,C 180,E1 -10978.009,E2 -10978.009} C_VEL
LIN {X 0,Y 404.315,Z 429.007,A -85,B 0,C 180,E1 -10979.004,E2 -10979.004} C_VEL
LIN {X 0,Y 404.229,Z 428.74,A -85,B 0,C 180,E1 -10980,E2 -10980} C_VEL
LIN {X 0,Y 404.243,Z 428.058,A -85,B 0,C 180,E1 -10980.996,E2 -10980.996} C_VEL
LIN {X 0,Y 404.165,Z 426.978,A -85,B 0,C 180,E1 -10981.993,E2 -10981.993} C_VEL
LIN {X 0,Y 404.277,Z 425.412,A -85,B 0,C 180,E1 -10982.99,E2 -10982.99} C_VEL
LIN {X 0,Y 404.251,Z 422.292,A -85,B 0,C 180,E1 -10984.487,E2 -10984.487} C_VEL
LIN {X 0,Y 404.5,Z 418.086,A -85,B 0,C 180,E1 -10985.984,E2 -10985.984} C_VEL
LIN {X 0,Y 404.831,Z 411.699,A -85,B 0,C 180,E1 -10987.732,E2 -10987.732} C_VEL
LIN {X 0,Y 405.113,Z 404.785,A -85,B 0,C 180,E1 -10989.234,E2 -10989.234} C_VEL
LIN {X 0,Y 405.577,Z 396.205,A -85,B 0,C 180,E1 -10990.736,E2 -10990.736} C_VEL
LIN {X 0,Y 406.01,Z 387.52,A -85,B 0,C 180,E1 -10991.989,E2 -10991.989} C_VEL
LIN {X 0,Y 406.574,Z 377.008,A -85,B 0,C 180,E1 -10993.241,E2 -10993.241} C_VEL
LIN {X 0,Y 407.143,Z 366.137,A -85,B 0,C 180,E1 -10994.3,E2 -10994.3} C_VEL
LIN {X 0,Y 407.538,Z 354.109,A -85,B 0,C 180,E1 -10995.247,E2 -10995.247} C_VEL
LIN {X 0,Y 408.013,Z 340.895,A -85,B 0,C 180,E1 -10996.062,E2 -10996.062} C_VEL
LIN {X 0,Y 408.358,Z 327.919,A -85,B 0,C 180,E1 -10996.658,E2 -10996.658} C_VEL
LIN {X 0,Y 408.688,Z 312.726,A -85,B 0,C 180,E1 -10997.127,E2 -10997.127} C_VEL
LIN {X 0,Y 410.664,Z 220.454,A -85,B 0,C 180,E1 -10999.207,E2 -10999.207} C_VEL
LIN {X 0,Y 407.389,Z 200.982,A -85,B 0,C 180,E1 -10999.842,E2 -10999.842} C_VEL
LIN {X 0,Y 408.708,Z 180.844,A -85,B 0,C 180,E1 -11003.566,E2 -11003.566} C_VEL
LIN {X 0,Y 408.978,Z 173.765,A -85,B 0,C 180,E1 -11004.898,E2 -11004.898} C_VEL
LIN {X 0,Y 406.325,Z 160.948,A -85,B 0,C 180,E1 -11007.56,E2 -11007.56} C_VEL
LIN {X 0,Y 404.174,Z 151.766,A -85,B 0,C 180,E1 -11009.556,E2 -11009.556} C_VEL
LIN {X 0,Y 404.147,Z 151.768,A -85,B 0,C 180,E1 -11012.621,E2 -11012.621} C_VEL
LIN {X 0,Y 404.186,Z 151.765,A -85,B 0,C 180,E1 -11015.189,E2 -11015.189} C_VEL
LIN {X 0,Y 404.152,Z 151.767,A -85,B 0,C 180,E1 -11018.757,E2 -11018.757} C_VEL
LIN {X 0,Y 404.123,Z 151.772,A -85,B 0,C 180,E1 -11021.598,E2 -11021.598} C_VEL
LIN {X 0,Y 404.15,Z 151.762,A -85,B 0,C 180,E1 -11024.521,E2 -11024.521} C_VEL
LIN {X 0,Y 404.141,Z 151.765,A -85,B 0,C 180,E1 -11027.295,E2 -11027.295} C_VEL
LIN {X 0,Y 404.174,Z 151.759,A -85,B 0,C 180,E1 -11029.955,E2 -11029.955} C_VEL
LIN {X 0,Y 404.14,Z 151.77,A -85,B 0,C 180,E1 -11033.125,E2 -11033.125} C_VEL
LIN {X 0,Y 404.149,Z 151.772,A -85,B 0,C 180,E1 -11036.187,E2 -11036.187} C_VEL
LIN {X 0,Y 404.169,Z 151.852,A -85,B 0,C 180,E1 -11039.21,E2 -11039.21} C_VEL
